500://Set home position and home flag
	IF Position <> DEFAULT_HOME_POSITION
	THEN
		MC_Home.Position									:= Position + (ABS(MemBlockPos - Axis.NcToPlc.ActPos) * SEL(MC_Velocity.Direction = MC_Negative_Direction, -1.0 , 1.0));
	ELSE
		MC_Home.Position									:= Param_CalibrationValue + (ABS(MemBlockPos - Axis.NcToPlc.ActPos) * SEL(MC_Velocity.Direction = MC_Negative_Direction, -1.0 , 1.0)); 
	END_IF
	MC_Home(
		Axis 		:= Axis,
		Execute		:= TRUE,
		Position	:= , //see above 
		HomingMode	:= MC_Direct
	);
	IF NOT MC_Home.Busy 
	THEN
		IF NOT MC_Home.Error
		THEN
			MemError										:= TRUE;
			LastErrorState									:= state;
			LastErrorId										:= MC_Absolute.ErrorID;	
			state											:= 600; //Try to restore old parameter first			
		ELSE
			state											:= 600;
		END_IF
		MC_Home(Execute := FALSE, Axis := Axis);
	END_IF

(* Return parameters for NC and drive to prior value ************************************************)
600:
	uiValue													:= TO_UINT(Param_MotionMonitoring.1);
	Write_ADS(NetId:= '' , Port:=500, IdxGrp:=16#4000+Axis.NcToPlc.AxisId, IDxOffs:=16#11,
				LEN:=SIZEOF(uiValue), SrcAddr:=ADR(uiValue), Write := Param_MotionMonitoring.0 );
	IF NOT Write_ADS.BUSY 
	THEN
		IF Write_ADS.ERR AND NOT MemError
		THEN
			MemError										:= TRUE;
			LastErrorState									:= state;
			LastErrorId										:= Write_ADS.ERRID;	
		END_IF
		Write_ADS(Write := FALSE);
		State												:= state + 1;									
	END_IF
		
601:
	uiValue													:= TO_UINT(Param_LagMonitoring.1);	
	Write_ADS(NetId:= '' , Port:=500, IdxGrp:=16#6000+Axis.NcToPlc.AxisId, IDxOffs:=16#10,
				LEN:=SIZEOF(uiValue), SrcAddr:=ADR(uiValue), Write := Param_LagMonitoring.0 );
	IF NOT Write_ADS.BUSY 
	THEN
		IF Write_ADS.ERR AND NOT MemError
		THEN
			MemError										:= TRUE;
			LastErrorState									:= state;
			LastErrorId										:= Write_ADS.ERRID;	
		END_IF
		Write_ADS(Write := FALSE);
		State												:= state + 1;									
	END_IF
	
602:
	uiValue													:= TO_UINT(Param_SoftMaxMonitoring.1);
	Write_ADS(NetId:= '' , Port:=500, IdxGrp:=16#5000+Axis.NcToPlc.AxisId, IDxOffs:=16#C,
				LEN:=SIZEOF(uiValue), SrcAddr:=ADR(uiValue), Write := Param_SoftMaxMonitoring.0 );
	IF NOT Write_ADS.BUSY 
	THEN
		IF Write_ADS.ERR AND NOT MemError
		THEN
			MemError										:= TRUE;
			LastErrorState									:= state;
			LastErrorId										:= Write_ADS.ERRID;	
		END_IF
		Write_ADS(Write := FALSE);
		State												:= state + 1;									
	END_IF
	
603:
	uiValue													:= TO_UINT(Param_SoftMinMonitoring.1);
	Write_ADS(NetId:= '' , Port:=500, IdxGrp:=16#5000+Axis.NcToPlc.AxisId, IDxOffs:=16#B,
				LEN:=SIZEOF(uiValue), SrcAddr:=ADR(uiValue), Write := Param_SoftMinMonitoring.0 );
	IF NOT Write_ADS.BUSY 
	THEN
		IF Write_ADS.ERR AND NOT MemError
		THEN
			MemError										:= TRUE;
			LastErrorState									:= state;
			LastErrorId										:= Write_ADS.ERRID;	
		END_IF
		Write_ADS(Write := FALSE);
		State												:= 604;									
	END_IF

604:
	IF DrvChannel = 1
	THEN
		CoERead.Index										:= SEL(DriveProfileIsDS402, 16#7110 , 	16#6872); 
		CoERead.SubIndex									:= SEL(DriveProfileIsDS402, 16#B  , 	16#0);
	ELSE //Channel 0
		CoERead.Index										:= SEL(DriveProfileIsDS402, 16#7010 , 	16#6072);
		CoERead.SubIndex									:= SEL(DriveProfileIsDS402, 16#B  , 	16#0);
 	END_IF 

	uiValue													:= Param_MaxTorque;
	CoEWrite(
		NetId			:= '', 
		Index			:= ,//See above
		SubIndex		:= , //See above 
		pSrcBuf			:= ADR(uiValue), 
		BufLen			:= SIZEOF(uiValue),//2,
		Execute			:= Param_MaxTorqueRead, 
		Axis			:= Axis
	);
	IF NOT CoEWrite.BUSY 
	THEN
		IF CoEWrite.Error
		THEN
			MemError										:= TRUE;
			LastErrorState									:= state;
			LastErrorId										:= CoEWrite.AdsErrId;//or CANopenErrId;				
		END_IF
		CoEWrite(Execute := FALSE, Axis := Axis);
		state												:= 900;			
	END_IF
	
(* Done *****************************************************************************)
900://Wait for execute signal to change to false
	Done 													:= NOT MemError; //Set the done flag to true if not error occur
	BUSY 													:= FALSE;
	Error													:= MemError;
	ErrorId													:= SEL(Error, 0 , LastErrorId);
	
	//Make sure all components stop operating
	Read_ADS(Read := FALSE);	Write_Ads(Write := FALSE);
	CoEWrite(Execute := FALSE,axis  := axis); CoERead(Execute := FALSE,axis  := axis);	
	MC_Home(Execute := FALSE,Axis := Axis);
	MC_Halt(Execute := FALSE,Axis := Axis);
	MC_Velocity(Execute := FALSE,Axis := Axis);
	MC_Absolute(Execute := FALSE,Axis := Axis);	
	
	State													:= 0;
END_CASE

END_FUNCTION_BLOCK

// POUs/Motion/TF50xx-NC/02_Options/Motion/AxMoveSinus
{attribute 'pack_mode' := '4'}
FUNCTION_BLOCK AxMoveSinus EXTENDS FbBase
VAR_INPUT
	Frequence												: LREAL := 0.0; //Hz
	SinusVeloAmplitude										: LREAL := 0.0; //mm/s
	DrivingTime												: TIME := T#0MS; //s
END_VAR
VAR_IN_OUT
	Axis													: AXIS_REF;
END_VAR
VAR_OUTPUT
	Active													: booL := FALSE;
	CommandAborted											: BOOL := FALSE;
END_VAR
VAR //Sinus Oscillation Sequence
(* 
- used as single sinus oscillation (sinus generator)
- used as sinus oscillation sequence (e.g. for bode plot) NEW 
UINT32 ENUM 1 				start type (fixed to start type 1 yet) 
UINT32 Reserved			
REAL64 e.g. mm/s > 0.0 		base amplitude (e.g. 2.5 mm/s) 
REAL64 Hz [0.0 .... 10.0] 	base frequency (e.g. 1.953125 Hz) 
REAL64 e.g. mm/s ≥ 0.0 		start amplitude at begin (e.g. 0.0 mm/s) 
REAL64 e.g. mm/REV > 0.0 	feed constant motor (per motor turn) (e.g. 10.0 mm/REV) 
REAL64 Hz ≥ 1.0 			frequency range: start frequency (e.g. 20.0 Hz) 
REAL64 Hz ≤ 1/(2*dT) 		frequency range: stop frequency (e.g. 500.0 Hz) 
REAL64 s > 0.0 				step duration (e.g. 2.048s) 
UINT32 1 [1 ... 200] 		number of measurements (step cycles) (e.g. 20) 
UINT32 1   					number of parallel measurements (e.g. 1)   not used yet! 
=72
*)   
	StartType												:	UDINT := TO_UDINT(Tc2_MC2._E_TCNC_StartPosType.TCNC_START_ABSOLUTE);
	Reserved												:	UDINT := 0;	
	BaseAmplitude											:	LREAL := 2.5;
	BaseFrequency											:	LREAL := 1.953125;
	StartAmplitude											:	LREAL := 0.0;
	FeedConstantMotor										:	LREAL := 10.0;
	FreqRangeStartFreq										:	LREAL := 0.0;
	FreqRangeStopFreq										:	LREAL := 500.0;								
	StepDuration											:	LREAL := 0.0;
	NumOfMeasurements										:	UDINT  := 0; //StepCount
	NumOfParallelMeasurements								:	UDINT  := 1;	
END_VAR
VAR
(* Internal memory **********************************************************************)
	LastErrorID												:	UDINT;
	StartCmdNo												: WORD;
	
(* Timer ********************************************************************************)                 	
	tonTimeout												:	TON;

(* Trigger ******************************************************************************)

(* FB instances *************************************************************************)
	Write_ADS												: ADSWRITE  := (NetId := '', Port := AMSPORT_R0_NCSAF, IdxGrp := 16#4200 + 0, IdxOffs := 16#33, LEN := 72, TmOut := DEFAULT_ADS_TIMEOUT);

(* Dummys *******************************************************************************)

END_VAR


(* Sinus Oscillation Sequence *************************************************************************************)
rtExecute(CLK := Execute);
CASE State OF
0://Wait for execute signal to change state to true
	IF NOT Execute OR rtExecute.Q	
	THEN
		Write_Ads(WRITE := FALSE);
		tonTimeout(IN := FALSE);
		FreqRangeStartFreq									:= Frequence;
		StartAmplitude										:= SinusVeloAmplitude;
		StepDuration										:= TO_LREAL(DrivingTime) * 0.001; //time ms to lreal s
		Busy												:= rtExecute.Q;
		CommandAborted										:= FALSE;
		Active												:= FALSE;
		Done 												:= FALSE;
		Error												:= FALSE;
		ErrorID												:= 0;
		StartCmdNo											:= Axis.NcToPlc.CmdNo;

		Write_ADS( //See also declaration
			IdxGrp	:=	16#4200+Axis.NcToPlc.AxisId,
			SrcAddr	:=ADR(StartType), 
			Write 	:= rtExecute.Q);
		
		state												:= SEL(Write_ADS.Write, 0, state + 1);
	
	END_IF

1://Read original parameters for position lag monitoring
	Write_ADS(SrcAddr	:=ADR(StartType)); 
	IF NOT Write_ADS.BUSY 
	THEN
		IF Write_ADS.ERR 
		THEN
			LastErrorId										:= Write_ADS.ERRID;	
			BUSY 											:= FALSE;
			Error											:= TRUE;
			ErrorId											:= LastErrorId;
			State											:= 0;
		ELSE				
			Active 											:= F_AxisHasJob(Axis.NcToPlc.StateDWord) AND StartCmdNo <> Axis.NcToPlc.CmdNo;	
			state											:= state + 1;
		END_IF
		Write_ADS(Write := FALSE);
	END_IF

2: //Wait for command done
	IF F_AxisHasJob(Axis.NcToPlc.StateDWord) AND StartCmdNo <> Axis.NcToPlc.CmdNo
	THEN
		Active												:= TRUE;
	ELSIF F_AxisInErrorState(Axis.NcToPlc.StateDWord) 
	THEN
		Active												:= FALSE;
		Busy												:= FALSE;
		(* axis error came up before this command has been started *)
		Error 												:= TRUE;
		ErrorID 											:= AXIS.NcToPlc.ErrorCode;
		LastErrorId											:= ErrorId;
		state												:= 0;
		
	ELSIF F_AxisIsCoupled(Axis.NcToPlc.CoupleState) 
		OR F_AxisHasBeenStopped(Axis.NcToPlc.StateDWord) 
	THEN
		(* if axis is coupled during motion (FlyingSaw) all commands are aborted *)
		Active												:= FALSE;
		Busy												:= FALSE;
		CommandAborted 										:= TRUE;
		state												:= 0;																																     	

	ELSIF Active
	THEN //No longer active
		Active												:= FALSE;
		Busy												:= FALSE;
		Done												:= TRUE;
		state												:= 0;		
	ELSE 	
		tonTimeOut(In := TRUE, PT := T#100MS);
		IF tonTimeOut.Q
		THEN //Command not responded
			Busy											:= FALSE;
			Error 											:= TRUE;
			ErrorID 										:= MC_ERROR_STATE_FEEDBACK_TIMEOUT;
			state											:= 0;				
		END_IF			
	END_IF
END_CASE
(********************************************************************************************)

END_FUNCTION_BLOCK

// POUs/Motion/TF50xx-NC/02_Options/Motion/AxSuperposition
FUNCTION_BLOCK AxSuperposition EXTENDS AxFbBase
VAR_OUTPUT CONSTANT 
	FNC_MOVEIMPOSED											:	INT := 0;
	FNC_MOVEABORT											:	INT := 1;
END_VAR                     								
VAR_INPUT                   								
	Fnc														:	INT := FNC_MOVEIMPOSED;
	Mode    												:	E_SuperpositionMode;
	Distance      											:	LREAL;
	VelocityDiff 											:	LREAL;
	Acc			 											:	LREAL;
	Dec			 											:	LREAL;
	Jerk    												:	LREAL;
	VelocityProcess   										:	LREAL;
	Length    												:	LREAL;
	Options    												:	ST_SuperpositionOptions;
                            							
END_VAR
VAR_IN_OUT
END_VAR
VAR_OUTPUT
	Warning													:	BOOL;
	WarningId												:	UDINT;
END_VAR
VAR
(* Zwischenspeicher ****************************************)
	MemFnc													:	INT := -1;

(* Timer ***************************************************)

(* Trigger *************************************************)

(* Instanzierung der MC Bausteine **************************)
	MC_MoveImposed											:	MC_MoveSuperImposed;
	MC_MoveAbort											:	MC_AbortSuperposition;

(* Dummy Speicher ******************************************)

END_VAR

	(************************************************************************************)
	(*																					*)
	(*		B E C K H O F F   N E W   A U T O M A T I O N   T E C H N O L O G Y    		*)
	(*																					*)
	(*		Eiserstr.5	D-33415 Verl	Germany	phone:	+49-5246-0	www.Beckhoff.com	*)
  	(*																					*)
  	(*		Bausteinbeschreibung	:	Move Imposed Achs Baustein						*)
	(*		TwinCAT-Version			:	3.1		 										*)
	(*		Version					:	V1.0 / 04/16									*)
 	(*																					*)
	(*																					*)
	(************************************************************************************)

(* Execute ******************************************************************************)
	rtExecute(CLK := Execute);
	IF rtExecute.Q
		AND MemFnc < 0
	THEN
		MemFnc 												:= Fnc ;
		Busy												:= TRUE;
		Done												:= FALSE;
		Active												:= FALSE;
		Error												:= FALSE;
		ErrorID												:= 0;
		Warning												:= FALSE;
		WarningId											:= 0;
		CmdAborted											:= FALSE;
		ErrorText											:= '';
	END_IF

(* Call Method ***********************************************************************************)
	CASE MemFnc OF
	FNC_MOVEIMPOSED:
		MoveImposed(Execute);

	FNC_MOVEABORT:
		MoveAbort(Execute);

	-1:
		IF NOT Execute
		THEN
			Busy											:= FALSE;
			Done											:= FALSE;
			Active											:= FALSE;
			Error											:= FALSE;
			ErrorID											:= 0;
			Warning											:= FALSE;
			WarningId										:= 0;
			CmdAborted										:= FALSE;
			ErrorText										:= '';
		END_IF
	ELSE
		Busy												:= FALSE;
		Done												:= FALSE;
		Active												:= FALSE;
		Error												:= Execute;
		ErrorID												:= E_AdsErr.DEVICE_INVALIDPARM;
		Warning												:= Execute;
		WarningId											:= 0;
		CmdAborted											:= FALSE;
		ErrorText											:= CONCAT('invalid parameter value(s) Fnc no: ' , INT_TO_STRING(MemFnc));
	END_CASE

(*************************************************************************************************)

METHOD PUBLIC moveAbort : BOOL //Return value = TRUE if busy
VAR_INPUT
	Execute													:	BOOL;
END_VAR
	MemFnc 													:= FNC_MOVEABORT;

IF NOT __ISVALIDREF(rAxis) 
THEN
	Busy													:= NOT Error;
	Error													:= TRUE;
	ErrorId													:= E_AdsErr.DEVICE_INVALIDPARM;
	CmdAborted												:= FALSE;
	Done													:= FALSE;
	Active													:= FALSE;
	ErrorText												:= 'Reference rAxis invalid (0)';
	MemFnc													:= SEL(Execute , -1 ,MemFnc); 
	RETURN;
END_IF


MC_MoveAbort(
	Execute													:= Execute,
	Axis													:= rAxis,
	Done													=> Done,
	Busy													=> Busy,
	Error													=> Error,
	ErrorID													=> ErrorID);

	IF Error THEN
		LastErrorId											:= ErrorID;
		ErrorText 											:= CONCAT('Error MC_MoveAbort ID:' , UDINT_TO_STRING(ErrorId));
	ELSE
		ErrorText 											:= '';
	END_IF

	IF NOT Execute AND NOT Busy
	THEN
		MemFnc												:=  -1;
	END_IF

	MoveAbort												:= Busy;
END_METHOD

METHOD PUBLIC moveImposed : BOOL //Return value = TRUE if busy
VAR_INPUT
	Execute													:	BOOL;
END_VAR
	MemFnc 													:= FNC_MOVEIMPOSED;
	
IF NOT __ISVALIDREF(rAxis) 
THEN
	Busy													:= NOT Error;
	Error													:= TRUE;
	ErrorId													:= E_AdsErr.DEVICE_INVALIDPARM;
	CmdAborted												:= FALSE;
	Done													:= FALSE;
	Active													:= FALSE;
	ErrorText												:= 'Reference rAxis invalid (0)';
	MemFnc													:= SEL(Execute , -1 ,MemFnc); 
	RETURN;
END_IF

	MC_MoveImposed(
		Execute												:= Execute,
		Mode												:= Mode,
		Distance											:= Distance,
		VelocityDiff										:= VelocityDiff,
		Acceleration										:= Acc,
		Deceleration										:= Dec,
		Jerk												:= Jerk,
		VelocityProcess										:= VelocityProcess,
		Length												:= Length,
		Options												:= Options,
		Axis												:= rAxis,
		Done												=> Done,
		Busy												=> Busy,
		Active												=> Active,
		CommandAborted										=> CmdAborted,
		Error												=> Error,
		ErrorID												=> ErrorID,
		Warning												=> Warning,
		WarningId											=> WarningID,
		ActualVelocityDiff									=> ,
		ActualDistance										=> ,
		ActualLength										=> ,
		ActualAcceleration									=> ,
		ActualDeceleration									=> );


	IF Error THEN
		LastErrorId											:= ErrorID;
		ErrorText 											:= CONCAT('Error MC_MoveSuperImposed ID:' , UDINT_TO_STRING(ErrorId));
	ELSE                            					
		ErrorText 											:= '';
	END_IF

	IF NOT Execute AND NOT Busy
	THEN
		MemFnc												:=  -1;
	END_IF

	MoveImposed												:= Busy;
END_METHOD

END_FUNCTION_BLOCK

// POUs/Motion/TF50xx-NC/02_Options/Parameter/AxParaCtrl
{attribute 'no_check'}
//FB to read and write NC axis controller parameter in particular  
//The FB can be enherided and derivatived methods of SeqRead/SeqWrite used for application specific parameter.
//The extended methods need to call the super class at the beginning and return true if execution will be finished. The allowed states for new parameter are 1..99
FUNCTION_BLOCK AxParaCtrl EXTENDS AxRWParaBase
VAR_OUTPUT CONSTANT
END_VAR                                 					
VAR_INPUT                               					                                   	                                        	
	AxisID													: 	UDINT;				(* ID der Achse *)

	(* Write *)
	SetPosLoopDeadBandPosDeviation							: 	LREAL;//Positon ctrl loop: 'dead band' in mm for position error (position deviation)(for P/PID-controller with velocity or torque interface)
	SetPosLoop_Kv											: 	LREAL;//Positon ctrl loop: Proportional amplification factor kp resp. kv (Standstill for two P-Const)
	SetPosLoop_Kv2Moving									: 	LREAL;//Positon ctrl loop: With two P-Const: Add proportional amplification factor kp resp. kv that applies above a limit velocity in percent 
	SetPosLoop_Tn											: 	LREAL;//Positon ctrl loop: Integral action time Tn in sec
	SetPosLoop_Tv											: 	LREAL;//Positon ctrl loop: Derivative action time Tv sec																			
	SetPosLoop_Td											: 	LREAL;//Positon ctrl loop: Damping time Td in sec																		
	
	SetPosLoopVeloThreshold									: 	LREAL;//Positon ctrl loop: Threshold level velocity in percent, above which the additional proportional amplification factor kp resp. kv applies.

	SetPosLoopMinMaxLimit_I_Part							: 	LREAL;//Positon ctrl loop: Min/Maximum output limitation ( ) for I- part in percent (default setting: 0.1 == 10 %)																	
	SetPosLoopMinMaxLimit_D_Part							: 	LREAL;//Positon ctrl loop: Min/Maximum output limitation ( ) for D- part in percent (default setting: 0.1 == 10 %)																
	SetPosLoopDisable_I_Part								: 	BOOL;//Positon ctrl loop: Switch off the I-part during an active positioning process (as far as I-part active)? (default setting: 0 = FALSE)										
 
	SetPosLoopFeedFwdAcc_Ka 								: 	LREAL;//Positon ctrl loop: Feed forward acceleration, proportional amplification factor Kv (Acceleration pre control)							
	SetPosLoopFeedFwdVeloPreCntrlWeight						: 	LREAL;//Positon ctrl loop: Weight of the velocity pre control (standard value: 1.0 = 100 %)
	
//Velocity control loop CtrlType 5,6)
	SetVeloLoopDeadBandVeloDeviation						: 	LREAL;//Velocity ctrl loop: 'dead band' for velocity error (velocity deviation)(for P/PID-controller with velocity or torque interface)
	SetVeloLoopFilterTimeVeloDeviation						: 	LREAL;//Velocity ctrl loop: PT-2 filter time for velocity error (velocity-difference)
                                                                         
	SetVeloLoop_Kv											: 	LREAL;//Velocity ctrl loop: The Proportional Factor Kv is the gain factor of the P-controller.
	SetVeloLoop_Tn											: 	LREAL;//Velocity ctrl loop: Integral Action Time Tn of the I component of the PID-controller in sec
	SetVeloLoop_Tv											: 	LREAL;//Velocity ctrl loop: Rate time Tv of the real D component (D-T1 component) of the PID-controller in sec																			
	SetVeloLoop_Td											: 	LREAL;//Velocity ctrl loop: Damping time Td of the real D component (D-T1 component) of the PID-controller in sec																		
                                                                         
	SetVeloLoopMinMaxLimit_D_Part							: 	LREAL;//Velocity ctrl loop: Min/Maximum output limitation ( ) for D- part in percent (default setting: 0.1 == 10 %)	
	SetVeloLoopMinMaxLimit_I_Part							: 	LREAL;//Velocity ctrl loop: Min/Maximum output limitation ( ) for I- part in percent (default setting: 0.1 == 10 %)																	

END_VAR
VAR_OUTPUT    
	CtrlType												: 	UDINT;(* Controller Type:
																			0 NOT DEFINED
																			1 Position-controller (standard) (Position)
																			2 Position-controller with two P-constants (with ka) (Position)
																			3 Position-controller PID (with ka)(Position)
																			5 Position and velocity P-controller(with ka) (Velocity)
																			6 PI controller (Velocity)
																			7 High/low speed controller (Position)
																			8 Stepper motor controller(Position)
																			9 SERCOS controller(Position in the drive)
																			10 RESERVED
																			11 RESERVED
																			12 RESERVED
																			13 RESERVED
																			14 TCom Controller (Soft Drive)(Position in the drive)*)

																		
//Position control loop
	PosLoopDeadBandPosDeviation								: 	LREAL;//Positon ctrl loop: 'dead band' in mm for position error (position deviation)(for P/PID-controller with velocity or torque interface)
	PosLoop_Kv												: 	LREAL;//Positon ctrl loop: Proportional amplification factor kp resp. kv (Standstill for two P-Const)
	PosLoop_Kv2Moving										: 	LREAL;//Positon ctrl loop: With two P-Const: Add proportional amplification factor kp resp. kv that applies above a limit velocity in percent 
	PosLoop_Tn												: 	LREAL;//Positon ctrl loop: Integral action time Tn in sec
	PosLoop_Tv												: 	LREAL;//Positon ctrl loop: Derivative action time Tv sec																			
	PosLoop_Td												: 	LREAL;//Positon ctrl loop: Damping time Td in sec																		
	
	PosLoopVeloThreshold									: 	LREAL;//Positon ctrl loop: Threshold level velocity in percent, above which the additional proportional amplification factor kp resp. kv applies.

	PosLoopMinMaxLimit_I_Part								: 	LREAL;//Positon ctrl loop: Maximum output limitation ( ) for I- part in percent (default setting: 0.1 == 10 %)																	
	PosLoopMinMaxLimit_D_Part								: 	LREAL;//Positon ctrl loop: Maximum output limitation ( ) for D- part in percent (default setting: 0.1 == 10 %)																
	PosLoopDisable_I_Part									: 	BOOL; //Positon ctrl loop: Switch off the I-part during an active positioning process (as far as I-part active)? (default setting: 0 = FALSE)										
 
	PosLoopFeedFwdAcc_Ka 									: 	LREAL;//Positon ctrl loop: Feed forward acceleration, proportional amplification factor Kv (Acceleration pre control)							
	PosLoopFeedFwdVeloPreCntrlWeight						: 	LREAL;//Positon ctrl loop: Weight of the velocity pre control (standard value: 1.0 = 100 %)

//Velocity control loop	(CtrlType 5,6)
	VeloLoopDeadBandVeloDeviation							: 	LREAL;//Velocity ctrl loop: 'dead band' for velocity error (velocity deviation)(for P/PID-controller with velocity or torque interface)
	VeloLoopFilterTimeVeloDeviation							: 	LREAL;//Velocity ctrl loop: PT-2 filter time for velocity error (velocity-difference)
                                                                          
	VeloLoop_Kv												: 	LREAL;//Velocity ctrl loop: The Proportional Factor Kv is the gain factor of the P-controller.
	VeloLoop_Tn												: 	LREAL;//Velocity ctrl loop: Integral Action Time Tn of the I component of the PID-controller in sec
	VeloLoop_Tv												: 	LREAL;//Velocity ctrl loop: Rate time Tv of the real D component (D-T1 component) of the PID-controller in sec																			
	VeloLoop_Td												: 	LREAL;//Velocity ctrl loop: Damping time Td of the real D component (D-T1 component) of the PID-controller in sec																		
                                                                         
	VeloLoopMinMaxLimit_D_Part								: 	LREAL;//Velocity ctrl loop: Min/Maximum output limitation ( ) for D- part in percent (default setting: 0.1 == 10 %)																
	VeloLoopMinMaxLimit_I_Part								: 	LREAL;//Velocity ctrl loop: Min/Maximum output limitation ( ) for I- part in percent (default setting: 0.1 == 10 %)																	
		
END_VAR                         	
VAR
(* Zwischenspeicher ************************************************************)
	
(* Deklaration Trigger **********************************************************)

(* Zeiten ******************************************************************)

(* Bausteine ***************************************************************)
	ReadAdsPara												: ADSREAD := (NetId	:= '' , Port := AMSPORT_R0_NC, TmOut	:= DEFAULT_ADS_TIMEOUT);
	WriteAdsPara											: ADSWRITE := (NetId:= '' , Port := AMSPORT_R0_NC, TmOut	:= DEFAULT_ADS_TIMEOUT);

(* Dummy Speicher **********************************************************)

END_VAR

	(************************************************************************************)
	(*																					*)
	(*		B E C K H O F F   N E W   A U T O M A T I O N   T E C H N O L O G Y    		*)
	(*																					*)
	(*		Eiserstr.5	D-33415 Verl	Germany	phone:	+49-5246-0	www.Beckhoff.Com	*)
    (*																					*)
    (*		Bausteinbeschreibung	:	Read/Write axis NC controller parameter			*)
	(*		TwinCAT-Version			:	3.x or higher									*)
	(*																					*)
	(************************************************************************************)

(* Execute ***************************************************************************************)
	Super^();			
	
(*************************************************************************************************)

PROPERTY PROTECTED deviceAddrIsValid : BOOL
GET
deviceAddrIsValid := AxisId > 0;
END_GET
END_PROPERTY

METHOD PROTECTED getValue : BOOL //Return value = TRUE if execution finished and state incremented 
VAR_INPUT
	IDxGrp						:	UDINT;
	IDxOffs						:	UDINT;
	Len							:	UDINT;
	pActValue					:	PVOID; //Address of variable for actual value
	pSetValue					:	PVOID; //Address of variable for ser value variable, can be zero if no corresponding SetVariable exists
END_VAR

ReadAdsPara	(Read := TRUE, IDxGrp:=IDxGrp+AxisId, IDxOffs:=IDxOffs,LEN:=Len,DestAddr:=pActValue );
IF NOT ReadAdsPara.BUSY
THEN
	IF NOT ReadAdsPara.ERR 
	THEN 
		IF pSetValue <> 0 THEN MEMCPY(pSetValue, pActValue, Len); END_IF			
		state 												:= state + 1; 
	ELSE 		
		Busy												:= FALSE;
		Error												:= TRUE;
		ErrorId												:= ReadAdsPara.ERRID;
		ErrorText											:= CONCAT('Error read parameter in state:' , TO_STRING(state * -1));
		ErrorText											:= CONCAT(ErrorText , ' Id:');
		ErrorText											:= CONCAT(ErrorText , TO_STRING(ErrorId));
		State												:= 9999;
	END_IF	
	ReadAdsPara(Read := FALSE); 
	getValue												:= TRUE;									
END_IF
END_METHOD

METHOD PROTECTED seqRead : BOOL //Return value = TRUE if execution finished 
VAR_IN_OUT
	State							:	INT;
END_VAR
(* Execute read axis parameter ************************************)
	CASE state OF
	1..99: //read application spec parameter 
		seqRead												:= TRUE;
		
	1001: (* Type **********************************************************************************)
		IF CtrlType <> 0 AND NOT ReadAdsPara.BUSY
		THEN
			state											:= state + 1;
		ELSE
			getValue(IDxGrp:= 16#6000,	IDxOffs := 16#3,	LEN := SIZEOF(CtrlType),	pActValue := ADR(CtrlType), 	pSetValue := 0);
		END_IF

	1002: (* Pos Ctrl loop. dead band (2,3,12,13 ****************************************************************************************)
		IF CtrlType <> 2 AND CtrlType <> 3 AND CtrlType <> 12 AND CtrlType <> 13 
		THEN
			state											:= state + 1;
		ELSE
			getValue(IDxGrp:= 16#6000,	IDxOffs := 16#10D,	LEN := SIZEOF(PosLoopDeadBandPosDeviation),	pActValue := ADR(PosLoopDeadBandPosDeviation), 	pSetValue := ADR(SetPosLoopDeadBandPosDeviation));
		END_IF

	1003: (* Pos control Kv (Standstill) (1,2,3,5,6,10,11,12,13 ****************************************************************************************)
		IF CtrlType > 6 AND CtrlType < 10 OR CtrlType > 13 
		THEN
			state											:= state + 1;
		ELSE
			getValue(IDxGrp:= 16#6000,	IDxOffs := 16#102,	LEN := SIZEOF(PosLoop_Kv),	pActValue := ADR(PosLoop_Kv), pSetValue := ADR(SetPosLoop_Kv));
		END_IF
		
	1004: (* Pos control Kv (Moving) (2, ****************************************************************************************)
		IF CtrlType <> 2 
		THEN
			state											:= state + 1;
		ELSE
			getValue(IDxGrp:= 16#6000,	IDxOffs := 16#106,	LEN := SIZEOF(PosLoop_Kv2Moving),	pActValue := ADR(PosLoop_Kv2Moving), pSetValue := ADR(SetPosLoop_Kv2Moving));
		END_IF
	
	1005: (* Pos control Integral action time Tn (3,10,11 ***********************************************************************)
		IF CtrlType <> 3 AND CtrlType <> 10 AND CtrlType <> 11
		THEN
			state											:= state + 1;
		ELSE
			getValue(IDxGrp:= 16#6000,	IDxOffs := 16#103,	LEN := SIZEOF(PosLoop_Tn),	pActValue := ADR(PosLoop_Tn),  pSetValue := ADR(SetPosLoop_Tn) );	
		END_IF
		
	1006: (* Pos control Derivative action time Tv (3,10,11 ***********************************************************************)
		IF CtrlType <> 3 AND CtrlType <> 10 AND CtrlType <> 11
		THEN
			state											:= state + 1;
		ELSE
			getValue(IDxGrp:= 16#6000,	IDxOffs := 16#104,	LEN := SIZEOF(PosLoop_Tv),	pActValue := ADR(PosLoop_Tv),  pSetValue := ADR(SetPosLoop_Tv) );
		END_IF
		
	1007: (* Pos control Damping time Td (3,10,11 ***************************************************************)
		IF CtrlType <> 3 AND CtrlType <> 10 AND CtrlType <> 11 
		THEN
			state											:= state + 1;
		ELSE
			getValue(IDxGrp:= 16#6000,	IDxOffs := 16#105,	LEN := SIZEOF(PosLoop_Td),	pActValue := ADR(PosLoop_Td), pSetValue := ADR(PosLoop_Td));
		END_IF

	1008: (* Pos control with 2 P-Const, Threshold level velocity in percent (2,) ***************************************************************)
		IF CtrlType <> 2 
		THEN
			state											:= state + 1;
		ELSE
			getValue(IDxGrp:= 16#6000,	IDxOffs := 16#107,	LEN := SIZEOF(PosLoopVeloThreshold),	pActValue := ADR(PosLoopVeloThreshold), pSetValue := ADR(SetPosLoopVeloThreshold));
		END_IF
		
	1009: (* Pos control Maximum output limitation ( ) for I- part in percent (3,10,11 ***************************************************************)
		IF CtrlType <> 3 AND CtrlType <> 10 AND CtrlType <> 11
		THEN
			state											:= state + 1;
		ELSE
			getValue(IDxGrp:= 16#6000,	IDxOffs := 16#116,	LEN := SIZEOF(PosLoopMinMaxLimit_I_Part),	pActValue := ADR(PosLoopMinMaxLimit_I_Part), pSetValue := ADR(SetPosLoopMinMaxLimit_I_Part));
		END_IF
		
	1010: (* Pos control Maximum output limitation ( ) for D- part in percent (3,10,11 ***************************************************************)
		IF CtrlType <> 3 AND CtrlType <> 10 AND CtrlType <> 11
		THEN
			state											:= state + 1;
		ELSE
			getValue(IDxGrp:= 16#6000,	IDxOffs := 16#117,	LEN := SIZEOF(PosLoopMinMaxLimit_D_Part),	pActValue := ADR(PosLoopMinMaxLimit_D_Part), pSetValue := ADR(SetPosLoopMinMaxLimit_D_Part));
		END_IF		

	1011: (* Pos control Switch off the I-part during an active positioning process (3,)***************************************************************)
		IF CtrlType <> 3 
		THEN
			state											:= state + 1;
		ELSIF getValue(IDxGrp:= 16#6000,	IDxOffs := 16#118,	LEN := SIZEOF(_UINT),	pActValue := ADR(_UINT),  pSetValue := 0)
		THEN
			SetPosLoopDisable_I_Part :=PosLoopDisable_I_Part := TO_BOOL(_UINT);
		END_IF
	
	1012:(* Pos control Feed forward acceleration (1,2,3,5,6,10,11,12,13 ***************************************************************)
		IF CtrlType > 6 AND CtrlType < 10 OR CtrlType > 13 
		THEN
			state											:= state + 1;
		ELSE
			getValue(IDxGrp:= 16#6000,	IDxOffs := 16#108,	LEN := SIZEOF(PosLoopFeedFwdAcc_Ka),	pActValue := ADR(PosLoopFeedFwdAcc_Ka), pSetValue := ADR(SetPosLoopFeedFwdAcc_Ka));
		END_IF	

	1013:(* Pos control Weight of the velocity pre contr *(1,2,3,5,6,10,11,12,13,14,..)  **************************************************************)
		getValue(IDxGrp:= 16#6000,	IDxOffs := 16#B,	LEN := SIZEOF(PosLoopFeedFwdVeloPreCntrlWeight),	pActValue := ADR(PosLoopFeedFwdVeloPreCntrlWeight), pSetValue := ADR(SetPosLoopFeedFwdVeloPreCntrlWeight));

//Velocity control 
	1014:(* Velocity control dead band velocity deviation (12, ***************************************************************)
		IF CtrlType <> 12
		THEN
			state											:= state + 1;
		ELSE
			getValue(IDxGrp:= 16#6000,	IDxOffs := 16#20D,	LEN := SIZEOF(VeloLoopDeadBandVeloDeviation),	pActValue := ADR(VeloLoopDeadBandVeloDeviation), pSetValue := ADR(SetVeloLoopDeadBandVeloDeviation));
		END_IF	
		
	1015:(* Velocity control Filter time velocity deviation (12, ***************************************************************)
		IF CtrlType <> 12
		THEN
			state											:= state + 1;
		ELSE
			getValue(IDxGrp:= 16#6000,	IDxOffs := 16#220,	LEN := SIZEOF(VeloLoopFilterTimeVeloDeviation),	pActValue := ADR(VeloLoopFilterTimeVeloDeviation), pSetValue := ADR(SetVeloLoopFilterTimeVeloDeviation));
		END_IF			
		
	1016:(* Velocity control: Proportional Factor Kv (5,6,12,13 ***************************************************************)
		IF CtrlType <> 5 AND CtrlType <> 6 AND CtrlType <> 12 AND CtrlType <> 13
		THEN
			state											:= state + 1;
		ELSE
			getValue(IDxGrp:= 16#6000,	IDxOffs := 16#202,	LEN := SIZEOF(VeloLoop_Kv),	pActValue := ADR(VeloLoop_Kv), pSetValue := ADR(SetVeloLoop_Kv));
		END_IF		
	
   	1017:(* Velocity control: Integral Action Time Tn (6,12***************************************************************)
		IF CtrlType <> 6 AND CtrlType <> 12
		THEN
			state											:= state + 1;
		ELSE
			getValue(IDxGrp:= 16#6000,	IDxOffs := 16#203,	LEN := SIZEOF(VeloLoop_Tn),	pActValue := ADR(VeloLoop_Tn), pSetValue := ADR(SetVeloLoop_Tn));
		END_IF										

   	1018:(* Velocity control: Derivative Action Time Tv (6,12 ***************************************************************)
		IF CtrlType <> 6 AND CtrlType <> 12
		THEN
			state											:= state + 1;
		ELSE
			getValue(IDxGrp:= 16#6000,	IDxOffs := 16#204,	LEN := SIZEOF(VeloLoop_Tv),	pActValue := ADR(VeloLoop_Tv), pSetValue := ADR(SetVeloLoop_Tv));
		END_IF	
		
   	1019:(* Velocity control: Damping Time Td (6,12 ***************************************************************)
		IF CtrlType <> 6 AND CtrlType <> 12
		THEN
			state											:= state + 1;
		ELSE
			getValue(IDxGrp:= 16#6000,	IDxOffs := 16#205,	LEN := SIZEOF(VeloLoop_Td),	pActValue := ADR(VeloLoop_Td), pSetValue := ADR(SetVeloLoop_Td));
		END_IF	
		
   	1020:(* Velocity control Min/Max limit I Part (6,12,13 ***************************************************************)
		IF CtrlType <> 6 AND CtrlType <> 12 AND CtrlType <> 13
		THEN
			state											:= state + 1;
		ELSE
			getValue(IDxGrp:= 16#6000,	IDxOffs := 16#206,	LEN := SIZEOF(VeloLoopMinMaxLimit_I_Part),	pActValue := ADR(VeloLoopMinMaxLimit_I_Part), pSetValue := ADR(SetVeloLoopMinMaxLimit_I_Part));
		END_IF	

   	1021:(* Velocity Min/max limit D Part (6,12 ***************************************************************)
		IF CtrlType <> 6 AND CtrlType <> 12
		THEN
			state											:= state + 1;
		ELSE
			getValue(IDxGrp:= 16#6000,	IDxOffs := 16#207,	LEN := SIZEOF(VeloLoopMinMaxLimit_D_Part),	pActValue := ADR(VeloLoopMinMaxLimit_D_Part), pSetValue := ADR(SetVeloLoopMinMaxLimit_D_Part));
		END_IF	
			
	ELSE
		state												:= 1;
	END_CASE

(*********************************************************************************************)
END_METHOD

METHOD PROTECTED seqWrite : BOOL //Return value = TRUE if execution finished 
VAR_IN_OUT
	State							:	INT;
END_VAR
(* Write axis parameter ********************************************************************)
	CASE state OF
	1..99: //Wite application spec parameter 
		seqWrite											:= TRUE;
			
	1001: (* Pos Ctrl loop. dead band  ****************************************************************************************)
		IF CtrlType <> 2 AND CtrlType <> 3 AND CtrlType <> 12 AND CtrlType <> 13 
		THEN
			state											:= state + 1;
		ELSE
			setValue(IDxGrp:= 16#6000,	IDxOffs := 16#10D,	LEN := SIZEOF(PosLoopDeadBandPosDeviation),	pActValue := ADR(PosLoopDeadBandPosDeviation), 	pSetValue := ADR(SetPosLoopDeadBandPosDeviation));
		END_IF

	1002: (* Pos control Kv (Standstill) ****************************************************************************************)
		IF CtrlType > 6 AND CtrlType < 10 OR CtrlType > 13 
		THEN
			state											:= state + 1;
		ELSE
			setValue(IDxGrp:= 16#6000,	IDxOffs := 16#102,	LEN := SIZEOF(PosLoop_Kv),	pActValue := ADR(PosLoop_Kv), pSetValue := ADR(SetPosLoop_Kv));
		END_IF
		
	1003: (* Pos control Kv (Moving) ****************************************************************************************)
		IF CtrlType <> 2 
		THEN
			state											:= state + 1;
		ELSE
			setValue(IDxGrp:= 16#6000,	IDxOffs := 16#106,	LEN := SIZEOF(PosLoop_Kv2Moving),	pActValue := ADR(PosLoop_Kv2Moving), pSetValue := ADR(SetPosLoop_Kv2Moving));
		END_IF
	
	1004: (* Pos control Integral action time Tn ***********************************************************************)
		IF CtrlType <> 3 AND CtrlType <> 10 AND CtrlType <> 11
		THEN
			state											:= state + 1;
		ELSE
			setValue(IDxGrp:= 16#6000,	IDxOffs := 16#103,	LEN := SIZEOF(PosLoop_Tn),	pActValue := ADR(PosLoop_Tn),  pSetValue := ADR(SetPosLoop_Tn) );	
		END_IF
		
	1005: (* Pos control Derivative action time Tv ***********************************************************************)
		IF CtrlType <> 3 AND CtrlType <> 10 AND CtrlType <> 11
		THEN
			state											:= state + 1;
		ELSE
			setValue(IDxGrp:= 16#6000,	IDxOffs := 16#104,	LEN := SIZEOF(PosLoop_Tv),	pActValue := ADR(PosLoop_Tv),  pSetValue := ADR(SetPosLoop_Tv) );
		END_IF
		
	1006: (* Pos control Damping time Td ***************************************************************)
		IF CtrlType <> 3 AND CtrlType <> 10 AND CtrlType <> 11
		THEN
			state											:= state + 1;
		ELSE
			setValue(IDxGrp:= 16#6000,	IDxOffs := 16#105,	LEN := SIZEOF(PosLoop_Td),	pActValue := ADR(PosLoop_Td), pSetValue := ADR(PosLoop_Td));
		END_IF

	1007: (* Pos control with 2 P-Const, Threshold level velocity in percent ***************************************************************)
		IF CtrlType <> 2 
		THEN
			state											:= state + 1;
		ELSE
			setValue(IDxGrp:= 16#6000,	IDxOffs := 16#107,	LEN := SIZEOF(PosLoopVeloThreshold),	pActValue := ADR(PosLoopVeloThreshold), pSetValue := ADR(SetPosLoopVeloThreshold));
		END_IF
		
	1008: (* Pos control Maximum output limitation ( ) for I- part in percent ***************************************************************)
		IF CtrlType <> 3 AND CtrlType <> 10 AND CtrlType <> 11
		THEN
			state											:= state + 1;
		ELSE
			setValue(IDxGrp:= 16#6000,	IDxOffs := 16#116,	LEN := SIZEOF(PosLoopMinMaxLimit_I_Part),	pActValue := ADR(PosLoopMinMaxLimit_I_Part), pSetValue := ADR(SetPosLoopMinMaxLimit_I_Part));
		END_IF
		
	1009: (* Pos control Maximum output limitation ( ) for D- part in percent ***************************************************************)
		IF CtrlType <> 3 AND CtrlType <> 10 AND CtrlType <> 11
		THEN
			state											:= state + 1;
		ELSE
			setValue(IDxGrp:= 16#6000,	IDxOffs := 16#117,	LEN := SIZEOF(PosLoopMinMaxLimit_D_Part),	pActValue := ADR(PosLoopMinMaxLimit_D_Part), pSetValue := ADR(SetPosLoopMinMaxLimit_D_Part));
		END_IF		

	1010: (* Pos control Switch off the I-part during an active positioning process ***************************************************************)
		IF NOT (SetPosLoopDisable_I_Part XOR PosLoopDisable_I_Part)
			AND NOT WriteAdsPara.BUSY
			OR CtrlType <> 3 
		THEN 
			state 											:= state + 1;
		ELSE
			_UINT											:= TO_UINT(SetPosLoopDisable_I_Part);
			PosLoopDisable_I_Part							:= SetPosLoopDisable_I_Part;
			setValue(IDxGrp:= 16#6000,	IDxOffs := 16#118,	LEN := SIZEOF(_UINT),		pActValue := 0,		pSetValue := ADR(_UINT));
		END_IF
		
	
	1011:(* Pos control Feed forward acceleration ***************************************************************)
		IF CtrlType > 6 AND CtrlType < 10 OR CtrlType > 13 
		THEN
			state											:= state + 1;
		ELSE
			setValue(IDxGrp:= 16#6000,	IDxOffs := 16#108,	LEN := SIZEOF(PosLoopFeedFwdAcc_Ka),	pActValue := ADR(PosLoopFeedFwdAcc_Ka), pSetValue := ADR(SetPosLoopFeedFwdAcc_Ka));
		END_IF	

	1012:(* Pos control Weight of the velocity pre contr ***************************************************************)
		setValue(IDxGrp:= 16#6000,	IDxOffs := 16#B,	LEN := SIZEOF(PosLoopFeedFwdVeloPreCntrlWeight),pActValue := ADR(PosLoopFeedFwdVeloPreCntrlWeight),	pSetValue := ADR(SetPosLoopFeedFwdVeloPreCntrlWeight));
		
//Velocity control 
	1013:(* Velocity control dead band velocity deviation ***************************************************************)
		IF CtrlType <> 12
		THEN
			state											:= state + 1;
		ELSE
			setValue(IDxGrp:= 16#6000,	IDxOffs := 16#20D,	LEN := SIZEOF(VeloLoopDeadBandVeloDeviation),	pActValue := ADR(VeloLoopDeadBandVeloDeviation), pSetValue := ADR(SetVeloLoopDeadBandVeloDeviation));
		END_IF	
		
	1014:(* Velocity control Filter time velocity deviation ***************************************************************)
		IF CtrlType <> 12
		THEN
			state											:= state + 1;
		ELSE
			setValue(IDxGrp:= 16#6000,	IDxOffs := 16#220,	LEN := SIZEOF(VeloLoopFilterTimeVeloDeviation),	pActValue := ADR(VeloLoopFilterTimeVeloDeviation), pSetValue := ADR(SetVeloLoopFilterTimeVeloDeviation));
		END_IF			
		
	1015:(* Velocity control: Proportional Factor Kv ***************************************************************)
		IF CtrlType <> 5 AND CtrlType <> 6 AND CtrlType <> 12 AND CtrlType <> 13
		THEN
			state											:= state + 1;
		ELSE
			setValue(IDxGrp:= 16#6000,	IDxOffs := 16#202,	LEN := SIZEOF(VeloLoop_Kv),	pActValue := ADR(VeloLoop_Kv), pSetValue := ADR(SetVeloLoop_Kv));
		END_IF		
	
   	1016:(* Velocity control: Integral Action Time Tn ***************************************************************)
		IF CtrlType <> 6 AND CtrlType <> 12
		THEN
			state											:= state + 1;
		ELSE
			setValue(IDxGrp:= 16#6000,	IDxOffs := 16#203,	LEN := SIZEOF(VeloLoop_Tn),	pActValue := ADR(VeloLoop_Tn), pSetValue := ADR(SetVeloLoop_Tn));
		END_IF										

   	1017:(* Velocity control: Derivative Action Time Tv ***************************************************************)
		IF  CtrlType <> 6 AND CtrlType <> 12
		THEN
			state											:= state + 1;
		ELSE
			setValue(IDxGrp:= 16#6000,	IDxOffs := 16#204,	LEN := SIZEOF(VeloLoop_Tv),	pActValue := ADR(VeloLoop_Tv), pSetValue := ADR(SetVeloLoop_Tv));
		END_IF	
		
   	1018:(* Velocity control: Damping Time Td ***************************************************************)
		IF CtrlType <> 6 AND CtrlType <> 12
		THEN
			state											:= state + 1;
		ELSE
			setValue(IDxGrp:= 16#6000,	IDxOffs := 16#205,	LEN := SIZEOF(VeloLoop_Td),	pActValue := ADR(VeloLoop_Td), pSetValue := ADR(SetVeloLoop_Td));
		END_IF	
		
   	1019:(* Velocity control Min/Max limit I Part ***************************************************************)
		IF CtrlType <> 6 AND CtrlType <> 12 AND CtrlType <> 13
		THEN
			state											:= state + 1;
		ELSE
			setValue(IDxGrp:= 16#6000,	IDxOffs := 16#206,	LEN := SIZEOF(VeloLoopMinMaxLimit_I_Part),	pActValue := ADR(VeloLoopMinMaxLimit_I_Part), pSetValue := ADR(SetVeloLoopMinMaxLimit_I_Part));
		END_IF	

   	1020:(* Velocity Min/max limit D Part ***************************************************************)
		IF CtrlType <> 6 AND CtrlType <> 12
		THEN
			state											:= state + 1;
		ELSE
			setValue(IDxGrp:= 16#6000,	IDxOffs := 16#207,	LEN := SIZEOF(VeloLoopMinMaxLimit_D_Part),	pActValue := ADR(VeloLoopMinMaxLimit_D_Part), pSetValue := ADR(SetVeloLoopMinMaxLimit_D_Part));
		END_IF	

	ELSE
		state 												:= 1 ;
	END_CASE
	
(***********************************************************************************************)
END_METHOD

METHOD PROTECTED setValue : BOOL //Return value = TRUE if execution finished and state incremented 
VAR_INPUT
	IDxGrp						:	UDINT;
	IDxOffs						:	UDINT;
	Len							:	UDINT;
	pActValue					:	PVOID; //Address of variable for actual value, can be zero if no corresponding acual value variable exists
	pSetValue					:	PVOID; //Address of variable for set value variable
END_VAR

IF pActValue <> 0 AND pSetValue <> 0 AND_THEN MEMCMP(pSetValue, pActValue, Len) = 0
THEN //Skip write parameter if set and actual value are equel
	state													:= state + 1;	
	setValue												:= TRUE;
ELSE
	WriteAdsPara( Write := TRUE, IdxGrp :=IDxGrp+AxisId, IdxOffs:=IDxOffs, LEN:=Len, SrcAddr:=pSetValue );
	IF NOT WriteAdsPara.BUSY
	THEN
		IF NOT WriteAdsPara.ERR
		THEN
			IF pActValue <> 0 THEN MEMCPY(pActValue, pSetValue, Len); END_IF	
			state											:= state + 1;
		ELSE
			Busy											:= FALSE;
			Error											:= TRUE;
			ErrorId											:= WriteAdsPara.ERRID;
			ErrorText										:= CONCAT('Error write parameter in state:' , TO_STRING(state * -1));
			ErrorText										:= CONCAT(ErrorText , ' Id:');
			ErrorText										:= CONCAT(ErrorText , TO_STRING(ErrorId));
			State											:= 9999;
		END_IF
		WriteAdsPara (Write := FALSE);
		setValue											:= TRUE;
	END_IF		
END_IF
END_METHOD

END_FUNCTION_BLOCK

// POUs/Motion/TF50xx-NC/02_Options/Phasing/AxPhasing
{attribute 'no_check'}
//Nc-axis phasing control 
//based on Tc2_MC2 library
FUNCTION_BLOCK AxPhasing EXTENDS AxFbBase
VAR_OUTPUT CONSTANT
	FNC_HALT_PHASING										:	INT := 0;
	FNC_PHASING_ABSOULTE									:	INT := 1;
	FNC_PHASING_RELATIVE									:	INT := 2;
END_VAR               
VAR_INPUT								
	Fnc														:	INT (FNC_HALT_PHASING..FNC_PHASING_RELATIVE) := FNC_HALT_PHASING;
	PhaseShift												:	LREAL := 0;
	Velo													:	LREAL := 0;
	Acc														:	LREAL := 0.0; // if Acc = 0, the NC-Value will be set                        								
	Dec														:	LREAL := 0.0; // if Dec = 0, the NC-Value will be set
	Jerk													:	LREAL := 0.0; // if Jerk = 0, the NC-Value will be set
	BufferMode												:	MC_BufferMode := MC_Aborting;(* 	MC_Aborting,
																									MC_Buffered,
																									MC_BlendingLow,
																									MC_BlendingPrevious,
																									MC_BlendingNext,
																									MC_BlendingHigh *)
                            								                        								
	Options 												: 	ST_PhasingOptions;
	rMasterAxis												:	REFERENCE TO AXIS_REF := 0;
END_VAR                     								
VAR_IN_OUT                  								
END_VAR                     									
VAR_OUTPUT                  	
	AbsolutePhaseShift										:	LREAL;
	CoveredPhaseShift										:	LREAL;
END_VAR
VAR
(* Zwischenspeicher **************************************************************************)
	MemFnc													:	INT := -1;

(* Trigger *)

(* Instanzierung der MC Bausteine *******************************************************)
	MC_HaltPhasing											:	MC_HaltPhasing;
	MC_PhasingAbsolute										:	MC_PhasingAbsolute;
	MC_PhasingRelative										:	MC_PhasingRelative;

(* Dummy Speicher **********************************************************)
(*	i,j		: INT := 0 ; *)
END_VAR

	(************************************************************************************)
	(*																					*)
	(*		B E C K H O F F   N E W   A U T O M A T I O N   T E C H N O L O G Y    		*)
	(*																					*)
	(*		Eiserstr.5	D-33415 Verl	Germany	phone:	+49-5246-0	www.Beckhoff.Com	*)
    (*																					*)
    (*		Bausteinbeschreibung	:	Gear axis function-block						*)
	(*		TwinCAT-Version			:	3.x or higher		 							*)
	(*		Version					:	V1.0 / 04/16									*)
 	(*		Autor					:	Thorsten Hemel									*)
	(*																					*)
	(************************************************************************************)

(* Execute ***************************************************************************************)
	rtExecute(CLK := Execute);
	IF rtExecute.Q
		AND MemFnc < 0
	THEN
		MemFnc 												:= Fnc ;
		Busy												:= TRUE;
		Done												:= FALSE;
		Active												:= FALSE;
		Error												:= FALSE;
		ErrorID												:= 0;
		CmdAborted											:= FALSE;
		ErrorText											:= '';
	END_IF

(* Call Method ***********************************************************************************)
	CASE MemFnc OF
	FNC_HALT_PHASING:
		HaltPhasing(Execute);

	FNC_PHASING_ABSOULTE:
		PhasingAbsoulte(Execute);

	FNC_PHASING_RELATIVE:
		PhasingRelative(Execute);

	-1:
		IF NOT Execute
		THEN
			Busy											:= FALSE;
			Done											:= FALSE;
			Active											:= FALSE;
			Error											:= FALSE;
			ErrorID											:= 0;
			CmdAborted										:= FALSE;
			ErrorText										:= '';
		END_IF                              				
	ELSE                                    				
		Busy												:= FALSE;
		Done												:= FALSE;
		Active												:= FALSE;
		Error												:= Execute;
		ErrorID												:= E_AdsErr.DEVICE_INVALIDPARM;
		CmdAborted											:= FALSE;
		ErrorText											:= CONCAT('invalid parameter value(s) Fnc no: ' , INT_TO_STRING(MemFnc));
	END_CASE                            		
                                            	

(*************************************************************************************************)

METHOD PUBLIC haltPhasing : BOOL //Return value = TRUE if busy
//required parameter
//rAxis
//rMasterAxis1
//RatioNumerator
//RatioDenominator
//Acc
//Dec
//Jerk
VAR_INPUT
	Execute													:	BOOL;
END_VAR
MemFnc 														:= FNC_HALT_PHASING;
THIS^.Execute												:= Execute;

IF NOT __ISVALIDREF(rAxis) 
THEN
	Busy													:= NOT Error;
	Error													:= TRUE;
	ErrorId													:= E_AdsErr.DEVICE_INVALIDPARM;
	CmdAborted												:= FALSE;
	Done													:= FALSE;
	Active													:= FALSE;
	ErrorText												:= 'Reference rAxis invalid (0)';
	MemFnc													:= SEL(Execute , -1 ,MemFnc); 
	RETURN;
ELSIF NOT __ISVALIDREF(rMasterAxis)
THEN
	Busy													:= NOT Error;
	Error													:= TRUE;
	ErrorId													:= E_AdsErr.DEVICE_INVALIDPARM;
	CmdAborted												:= FALSE;
	Done													:= FALSE;
	ErrorText												:= 'Reference rMasterAxis invalid (0)';
	MemFnc													:= SEL(Execute , -1 ,MemFnc); 
	RETURN;
END_IF

	MC_HaltPhasing(
		Execute				:= Execute, 
		Master				:= rMasterAxis, 
		Slave				:= rAxis, 
		Deceleration		:= Dec, 
		Jerk				:= Jerk, 
		BufferMode			:= BufferMode, 
		Options				:= Options, 
		Done				=> Done, 
		Busy				=> Busy, 
		Active				=> Active, 
		CommandAborted		=> CmdAborted, 
		Error				=> Error, 
		ErrorID				=> ErrorID);

	IF Error THEN
		LastErrorId											:= ErrorID;
		ErrorText 											:= CONCAT('Error MC_HaltPhasing ID:' , UDINT_TO_STRING(ErrorId));
	ELSE
		ErrorText 											:= '';
	END_IF

	IF NOT Execute AND NOT Busy
	THEN
		MemFnc												:=  -1;
	END_IF
	
	haltPhasing												:= Busy;
END_METHOD

METHOD PUBLIC phasingAbsoulte : BOOL //Return value = TRUE if busy
//required parameter
//rAxis
//rMasterAxis
//PhaseShift
//Acc
VAR_INPUT
	Execute													:	BOOL;
END_VAR
MemFnc 														:= FNC_PHASING_ABSOULTE;
THIS^.Execute												:= Execute;

IF NOT __ISVALIDREF(rAxis) 
THEN
	Busy													:= NOT Error;
	Error													:= TRUE;
	ErrorId													:= E_AdsErr.DEVICE_INVALIDPARM;
	CmdAborted												:= FALSE;
	Done													:= FALSE;
	Active													:= FALSE;
	ErrorText												:= 'Reference rAxis invalid (0)';
	MemFnc													:= SEL(Execute , -1 ,MemFnc); 
	RETURN;
ELSIF NOT __ISVALIDREF(rMasterAxis)
THEN
	Busy													:= NOT Error;
	Error													:= TRUE;
	ErrorId													:= E_AdsErr.DEVICE_INVALIDPARM;
	CmdAborted												:= FALSE;
	Done													:= FALSE;
	ErrorText												:= 'Reference rMasterAxis1 invalid (0)';
	MemFnc													:= SEL(Execute , -1 ,MemFnc); 
	RETURN;
END_IF

	MC_PhasingAbsolute(
		Execute				:= Execute, 
		Master				:= rMasterAxis, 
		Slave				:= rAxis, 
		PhaseShift			:= PhaseShift, 
		Velocity			:= Velo, 
		Acceleration		:= Acc, 
		Deceleration		:= Dec, 
		Jerk				:= Jerk, 
		BufferMode			:= BufferMode, 
		Options				:= Options, 
		Done				=> Done, 
		Busy				=> Busy, 
		Active				=> Active, 
		CommandAborted		=> CmdAborted, 
		Error				=> Error, 
		ErrorID				=> ErrorId, 
		AbsolutePhaseShift	=> AbsolutePhaseShift);
		

	IF Error THEN
		LastErrorId											:= ErrorID;
		ErrorText 											:= CONCAT('Error MC_PhasingAbsolute ID:' , UDINT_TO_STRING(ErrorId));
	ELSE
		ErrorText 											:= '';
	END_IF

	IF NOT Execute AND NOT Busy
	THEN
		MemFnc												:=  -1;
	END_IF
	
	phasingAbsoulte											:= Busy;
END_METHOD

METHOD PUBLIC phasingRelative : BOOL//Return value = TRUE if busy
//required parameter
//rAxis
//rMasterAxis
//PhaseShift
//Acc
VAR_INPUT
	Execute													:	BOOL;
END_VAR
MemFnc														:= FNC_PHASING_RELATIVE;
THIS^.Execute												:= Execute;
	                										
IF NOT __ISVALIDREF(rAxis) 
THEN
	Busy													:= NOT Error;
	Error													:= TRUE;
	ErrorId													:= E_AdsErr.DEVICE_INVALIDPARM;
	CmdAborted												:= FALSE;
	Done													:= FALSE;
	Active													:= FALSE;
	ErrorText												:= 'Reference rAxis invalid (0)';
	MemFnc													:= SEL(Execute , -1 ,MemFnc); 
	RETURN;
ELSIF NOT __ISVALIDREF(rMasterAxis)
THEN
	Busy													:= NOT Error;
	Error													:= TRUE;
	ErrorId													:= E_AdsErr.DEVICE_INVALIDPARM;
	CmdAborted												:= FALSE;
	Done													:= FALSE;
	ErrorText												:= 'Reference rMasterAxis invalid (0)';
	MemFnc													:= SEL(Execute , -1 ,MemFnc); 
	RETURN;	
END_IF
	

	MC_PhasingRelative( 
		Execute				:= Execute,
		Master				:= rMasterAxis, 
		Slave				:= rAxis, 
		PhaseShift			:= PhaseShift, 
		Velocity			:= Velo, 
		Acceleration		:= Acc, 
		Deceleration		:= Dec, 
		Jerk				:= Jerk, 
		BufferMode			:= BufferMode, 
		Options				:= Options, 
		Done				=> Done, 
		Busy				=> Busy, 
		Active				=> Active, 
		CommandAborted		=> CmdAborted, 
		Error				=> Error, 
		ErrorID				=> ErrorId, 
		CoveredPhaseShift	=> CoveredPhaseShift);					

	IF Error THEN
		LastErrorId											:= ErrorID;
		ErrorText 											:= CONCAT('Error MC_PhasingRelative ID:' , UDINT_TO_STRING(ErrorId));
	ELSE
		ErrorText 											:= '';
	END_IF

	IF NOT Execute AND NOT Busy
	THEN
		MemFnc												:=  -1;
	END_IF
	
	phasingRelative												:= Busy;
END_METHOD

END_FUNCTION_BLOCK

// POUs/Motion/TF50xx-NC/02_Options/TouchProbe/AxTouchProbe
{attribute 'no_check'}
//Nc-axis touch probe  
//based on Tc2_MC2 library
FUNCTION_BLOCK AxTouchProbe EXTENDS AxFbBase
VAR_OUTPUT CONSTANT
	FNC_RUN													:	INT := 0;
	FNC_ABORT												:	INT := 1;
END_VAR                     								
VAR_INPUT                   								
	Fnc														: 	INT (FNC_RUN..FNC_ABORT):= FNC_RUN;
	TriggerInput											: 	TRIGGER_REF;
	WindowOnly												: 	BOOL := FALSE;(* Enables the monitoring window *)
	FirstPosition											: 	LREAL;	(* Beginning of the monitoring window *)
	LastPosition 											: 	LREAL;	(* Ending of the monitoring window *)
END_VAR
VAR_IN_OUT
END_VAR
VAR_OUTPUT
	RecordedPosition										: 	LREAL;	// current axisposition on trigger-event
	RecordedData											:	MC_TouchProbeRecordedData;
END_VAR
VAR
(* cache **************************************************************************)
	MemFnc													:	INT := -1;
               								                           	
(* trigger *)               	

(* MC-function-block instances ****************************************************)
	MC_TouchProbe											: 	MC_TouchProbe;
	MC_AbortTrigger											:	MC_AbortTrigger;

END_VAR

	(************************************************************************************)
	(*																					*)
	(*		B E C K H O F F   N E W   A U T O M A T I O N   T E C H N O L O G Y    		*)
	(*																					*)
	(*		Eiserstr.5	D-33415 Verl	Germany	phone:	+49-5246-0	www.Beckhoff.Com	*)
    (*																					*)
    (*		Bausteinbeschreibung	:	TouchProbe ctrl									*)
	(*		TwinCAT-Version			:	3.x or higher 									*)
	(*		Version					:	V3.0 / 03/13									*)
	(*		Lib						:	TcMC2.lib 										*)
 	(*		Autor					:	DSC												*)
	(*																					*)
	(************************************************************************************)

(* Execute ***************************************************************************************)
	rtExecute(CLK := Execute);
	IF rtExecute.Q
		AND MemFnc < 0
	THEN
		MemFnc 												:= SEL(Fnc = FNC_RUN, FNC_ABORT , FNC_RUN) ;
		Busy												:= TRUE;
		Done												:= FALSE;
		Error												:= FALSE;
		ErrorID												:= 0;
		CmdAborted											:= FALSE;
	END_IF

(* Call Method ***********************************************************************************)
	CASE MemFnc OF
	FNC_RUN:
		Run(Execute);

	FNC_ABORT:
		Abort(Execute);

	-1:
		IF NOT Execute
		THEN
			Busy											:= FALSE;
			Done											:= FALSE;
			Error											:= FALSE;
			ErrorID											:= 0;
			CmdAborted										:= FALSE;
		END_IF                              				
	ELSE                                    				
		Busy												:= FALSE;
		Done												:= FALSE;
		Error												:= Execute;
		ErrorID												:= E_AdsErr.DEVICE_INVALIDPARM;
		CmdAborted											:= FALSE;
	END_CASE                                	

(*************************************************************************************************)

METHOD PUBLIC abort : BOOL //Return value = TRUE if busy
//required parameter
//rAxis
//TriggerInput
VAR_INPUT
	Execute													:	BOOL := FALSE;
END_VAR
	MemFnc	 												:= FNC_ABORT;
	THIS^.Execute											:= Execute;
IF NOT __ISVALIDREF(rAxis) 
THEN
	Busy													:= NOT Error;
	ErrorId													:= E_AdsErr.DEVICE_INVALIDPARM;
	Error													:= TRUE;
	Done													:= FALSE;
	CmdAborted												:= FALSE;
	MemFnc													:= SEL(Execute , -1 ,MemFnc); 
	RETURN;
END_IF

	MC_AbortTrigger(
		Execute		:= Execute,
		Axis		:= rAxis,
		TriggerInput:= TriggerInput,
		Done		=> done,
		Busy		=> Busy,
		Error		=> Error,
		ErrorID		=> ErrorID);

	CmdAborted		:= FALSE;

	IF NOT Execute AND NOT Busy
	THEN
		MemFnc												:= -1;
	END_IF                              					
	                                    	
	abort 													:= Busy;
END_METHOD

METHOD PUBLIC run : BOOL //Return value = TRUE if busy
//required parameter
//rAxis
//TriggerInput
//WindowOnly
//FirstPosition
//LastPosition
VAR_INPUT
	Execute													: BOOL := FALSE;
END_VAR
	MemFnc 													:= FNC_RUN;
	THIS^.Execute											:= Execute;
	
IF NOT __ISVALIDREF(rAxis) 
THEN
	Busy													:= NOT Error;
	ErrorId													:= E_AdsErr.DEVICE_INVALIDPARM;
	Error													:= TRUE;
	Done													:= FALSE;
	CmdAborted												:= FALSE;
	MemFnc													:= SEL(Execute , -1 ,MemFnc); 
	RETURN;
END_IF

	MC_TouchProbe(
		Execute			:= Execute,
		WindowOnly		:= WindowOnly,
		FirstPosition	:= FirstPosition,
		LastPosition	:= LastPosition,
		Axis			:= rAxis,
		TriggerInput	:= TriggerInput,
		Done			=> Done,
		Busy			=> Busy,
		CommandAborted	=> CmdAborted,
		Error			=> Error,
		ErrorID			=> ErrorID,
		RecordedPosition=> RecordedPosition,
		RecordedData 	=> RecordedData);

	IF NOT Execute AND NOT Busy
	THEN
		MemFnc												:= -1;
	END_IF
	
	run														:= busy;
END_METHOD

END_FUNCTION_BLOCK

// POUs/Motion/TF50xx-NC/03_Utilities/AX_JOB
FUNCTION_BLOCK AX_JOB (* Datatyp/Object - Ax Start data *)
VAR_INPUT
//	name						:	STRING(10);
	Fnc														:	INT := 0;
	BufferMode												:	MC_BufferMode := MC_Aborting;(* 	MC_Aborting,
																									MC_Buffered,
																									MC_BlendingLow,
																									MC_BlendingPrevious,
																									MC_BlendingNext,
																									MC_BlendingHigh *)
	Direction												:	MC_Direction := MC_POSITIVE_DIRECTION;	(*	MC_POSITIVE_DIRECTION,
																						   					MC_SHORTeSTATE.WAY,
																						   					MC_NEGATIVE_DIRECTION,
																						   					MC_CURRENT_DIRECTION *)
	Target													:	LREAL	:= 0.0; // target position
	Velo													: 	LREAL	:= 0.0; // target velocity mm/s
	Override												:	LREAL := 100.0; // override
	Acc														:	LREAL := 0.0; // acceleration
	Dec														:	LREAL := 0.0; // deceleration
	Jerk													:	LREAL := 0.0; // jerk
	InTarget												:	BOOL := FALSE;
	InPosWindow												:	BOOL := FALSE;
END_VAR
VAR_OUTPUT
END_VAR
VAR
END_VAR

;

METHOD PUBLIC reset : BOOL
VAR_INPUT
END_VAR
Fnc															:= 0;
BufferMode													:= MC_Aborting;
Direction													:= MC_CURRENT_DIRECTION;
Target														:= 0;
Velo														:= 0;
Override													:= 0;
InTarget													:= FALSE;
InPosWindow													:= FALSE;
reset														:= TRUE;
END_METHOD

END_FUNCTION_BLOCK

// POUs/Motion/TF50xx-NC/03_Utilities/AxAutoFct
{attribute 'no_check'}
FUNCTION_BLOCK AxAutoFct
VAR_INPUT
	Enable													:	BOOL := FALSE;(* Enable block *)
	AutoInit												:	BOOL := TRUE; (* TRUE=With Enable force status will be written to axis / FALSE=Force values will only be written on change *) 
	AxisId													: 	DWORD; (* ID der Achse *)
	ForceSoftLimit											:	BOOL := TRUE; (* TRUE => SoftLimitMonitoring = True *)
	ForceCalibration										:	BOOL := FALSE;(* TRUE => Calibrated = True  *)
	ForcePosLagMon											:	BOOL := TRUE; (* TRUE => Position Lag Monitoring = True  *)
	ForcePosMon												:	BOOL := TRUE; (* TRUE => In Position Monitoring = True  *)
	ForceTargetMon											:	BOOL := TRUE; (* TRUE => In Target Monitoring = True  *)
END_VAR                         							
VAR_IN_OUT                      							
END_VAR                         							
VAR_OUTPUT        
	{attribute 'displaymode':='binary'}              							
	Status													:	BYTE := 0;
	Busy													:	BOOL := FALSE;
	Error													:	BOOL := FALSE;
	ErrorID													:	UDINT := 0;
END_VAR                         	

VAR
(* Cache **********************************************************************)
	State													: 	INT;
	InitDone												:	BYTE;
	LastErrText												:	STRING(20);
	
(* Instances *******************************************************************)
	WriteAdsPara											: 	ADSWRITE := (NetID:= '' , Port:=AMSPORT_R0_NC, TmOut	:= DEFAULT_ADS_TIMEOUT);

(* Dummy  *********************************************************************)
	tmpWORD													:	UINT;

END_VAR

	(* Enable/Disable of: Soft limit monitoring, Target monitoring, Pos. Lag monitoring,  Calibration 	*)
	(*																									*)
	(****************************************************************************************************)

(* writing parameters *******************************************************************************)
IF NOT Enable 
THEN
	Status.0 												:= NOT forceSoftLimit;
	Status.1 												:= NOT forceCalibration;
	Status.2 												:= NOT forcePosLagMon;
	Status.3 												:= NOT forcePosMon;
	Status.4 												:= NOT forceTargetMon;
	            											
	InitDone 												:= SEL(AutoInit , 2#0001_1111 , 2#0000_0000);
                											
	State 													:= 0;
	Error													:= FALSE;
	ErrorID													:= 0;
	Busy 													:= FALSE;
ELSIF AxisId = 0 
THEN
	ErrorID													:= E_AdsErr.DEVICE_INVALIDPARM;
	Error													:= FALSE;
	Busy													:= FALSE;
ELSE
	CASE State OF
	0:	(* Init *)

		Busy := FALSE;

		IF NOT WriteAdsPara.BUSY
			AND NOT WriteAdsPara.WRITE
		 	AND NOT Error
		THEN
			IF (forceSoftLimit XOR status.0) OR NOT InitDone.0 THEN
				InitDone.0 									:= TRUE;
				status.0 									:= forceSoftLimit;
				tmpWord 									:= BOOL_TO_UINT(forceSoftLimit);
				State 										:= 1;
				Busy 										:= TRUE;

			ELSIF(forceCalibration XOR status.1) OR NOT InitDone.1 THEN
				InitDone.1 									:= TRUE;
				status.1 									:= forceCalibration;
				tmpWord 									:= BOOL_TO_UINT(forceCalibration);
				State 										:= 10;
				Busy 										:= TRUE;
	
			ELSIF(forcePosLagMon XOR status.2) OR NOT InitDone.2 THEN
				InitDone.2 									:= TRUE;
				status.2 									:= forcePosLagMon;
				tmpWord 									:= BOOL_TO_UINT(forcePosLagMon);
				State 										:= 20;
				Busy 										:= TRUE;
			ELSIF(forcePosMon XOR status.3) OR NOT InitDone.3 THEN
				InitDone.3 									:= TRUE;
				status.3 									:= forcePosMon;
				tmpWord 									:= BOOL_TO_UINT(forcePosMon);
				State 										:= 30;
				Busy 										:= TRUE;
			ELSIF(forceTargetMon XOR status.4) OR NOT InitDone.4 THEN
				InitDone.4 									:= TRUE;
				status.4 									:= forceTargetMon;
				tmpWord 									:= BOOL_TO_UINT(forceTargetMon);
				State 										:= 40;
				Busy 										:= TRUE;
		
			END_IF
		ELSE
			WriteAdsPara	(Write := FALSE);
		END_IF

	1: (* toggle positive limit switches ****************************************************************)
		IF NOT WriteAdsPara.Busy
			AND WriteAdsPara.Write
		THEN
			IF WriteAdsPara.Err THEN
				State 										:= 9999;  // goto Error-state 
			ELSE           									
				State 										:= State + 1;
			END_IF         	
		END_IF

		WriteAdsPara(
			IdxGrp	:=16#4000+AxisId,
			IdxOffs	:=16#1000C,
			LEN		:=SIZEOF(tmpWord),
			SrcAddr	:=ADR(tmpWord),
			Write 	:= State = 1);

	2: (* toggle negative limit switches *****************************************************************)
		IF NOT WriteAdsPara.Busy
			AND WriteAdsPara.Write
		THEN
			IF WriteAdsPara.Err THEN
				State 										:= 9999; // goto Error-state 
			ELSE
				State 										:= 99; // done 
			END_IF
		END_IF

		WriteAdsPara(
			IdxGrp	:=16#4000+AxisId,
			IdxOffs	:=16#1000B,
			LEN		:=SIZEOF(tmpWord),
			SrcAddr	:=ADR(tmpWord),
			Write 	:= State = 2);

	10: (* set referenceflag *****************************************************************)
		IF NOT WriteAdsPara.Busy
			AND WriteAdsPara.Write
		THEN
			IF WriteAdsPara.Err THEN
				State 										:= 9999;  	// goto Error-state 
			ELSE           									
				State 										:= 99; 		// done 
			END_IF
		END_IF

		WriteAdsPara(
			IdxGrp	:=16#5100+AxisId,
			IdxOffs	:=16#9,
			LEN		:=SIZEOF(tmpWord),
			SrcAddr	:=ADR(tmpWord),
			Write 	:= State = 10 );
			
	20: (* lagdistance monitoring *****************************************************************)
		IF NOT WriteAdsPara.Busy
			AND WriteAdsPara.Write
		THEN
			IF WriteAdsPara.Err THEN
				State 										:= 9999;  	// goto Error-state 
			ELSE           									
				State 										:= 99; 		// done
			END_IF
		END_IF

		WriteAdsPara(
			IdxGrp	:=16#6000+AxisId,
			IdxOffs	:=16#10,
			LEN		:=SIZEOF(tmpWord),
			SrcAddr	:=ADR(tmpWord),
			Write 	:= State = 20);
			
	30: (* Position Monitoring *****************************************************************)
		IF NOT WriteAdsPara.Busy
			AND WriteAdsPara.Write
		THEN
			IF WriteAdsPara.Err THEN
				State 										:= 9999;  	// goto Error-state 
			ELSE           									
				State 										:= 99; 		// done
			END_IF
		END_IF

		WriteAdsPara(

			IdxGrp	:=16#4000+AxisId,
			IdxOffs	:=16#F,
			LEN		:=SIZEOF(tmpWord),
			SrcAddr	:=ADR(tmpWord),
			Write 	:= State = 30 );

	40: (* Target Monitoring *****************************************************************)
		IF NOT WriteAdsPara.Busy
			AND WriteAdsPara.Write
		THEN
			IF WriteAdsPara.Err THEN
				State 										:= 9999;  	// goto Error-state 
			ELSE           									
				State 										:= 99; 		// done
			END_IF
		END_IF

		WriteAdsPara(
			IdxGrp	:=16#4000+AxisId,
			IdxOffs	:=16#15,
			LEN		:=SIZEOF(tmpWord),
			SrcAddr	:=ADR(tmpWord),
			Write 	:= State = 40 );
			
	ELSE (* case else *)
		IF WriteAdsPara.ERR THEN
			Error											:= TRUE;
			ErrorID											:= WriteAdsPara.ERRID;
			LastErrText										:= CONCAT('Err WriteAdsPara ID: ', UDINT_TO_STRING(ErrorID));
		ELSE            									
			State 											:= 0;
		END_IF
	END_CASE
END_IF

(************************************************************************************************************************)

END_FUNCTION_BLOCK

// POUs/Motion/TF50xx-NC/03_Utilities/AxAutoWriteSoftLimit
{attribute 'no_check'}
FUNCTION_BLOCK AxAutoWriteSoftLimit
VAR_INPUT
	Enable													:	BOOL := FALSE; (* Enable Block *)
	AxId													: 	DWORD; (* ID der Achse *)
	SoftLimitPos											:	LREAL;
	SoftLimitNeg											:	LREAL;
END_VAR                         							
VAR_IN_OUT                      							
END_VAR                         							
VAR_OUTPUT        
	Busy													:	BOOL := FALSE;
	Error													:	BOOL := FALSE;
	{attribute 'displaymode':='hex'}  
	ErrorID													:	UDINT := 0;
END_VAR                         	
VAR
(* Cache **********************************************************************)
	State													: 	INT;
	MemLimitPos												:	LREAL;
	MemLimitNeg												:	LREAL;
	WriteReg												:	BYTE;

(* Instances *******************************************************************)
	WriteAdsPara											: 	ADSWRITE := (NetId	:= '' , Port := 500, TmOut	:= DEFAULT_ADS_TIMEOUT);

(* Dummy  *********************************************************************)
END_VAR

	(* Easy soft limit change 																		*)
	(************************************************************************************************)

(* writing parameters *******************************************************************************)
IF NOT Enable 
THEN
	MemLimitPos												:= SoftLimitPos;
	MemLimitNeg												:= SoftLimitNeg;
	                										
	State 													:= 0;
	Error													:= FALSE;
	ErrorID													:= 0;
	Busy 													:= FALSE;
ELSIF Axid = 0 
THEN
	ErrorID													:= E_AdsErr.DEVICE_INVALIDPARM;
	Error													:= FALSE;
	Busy													:= FALSE;
ELSE
	CASE State OF
	0:	(* Init *)

		Busy 												:= FALSE;

		IF NOT WriteAdsPara.BUSY
			AND NOT WriteAdsPara.WRITE
		 	AND NOT Error
		THEN
			WriteReg.0										:= SoftLimitPos <> MemLimitPos;
			WriteReg.1										:= SoftLimitNeg <> MemLimitNeg;
			
			IF WriteReg <> 0
			THEN
				Busy 										:= TRUE;
				state										:= state + SEL(WriteReg.0, 2, 1); //Jump to 2 if only negative changed
				MemLimitPos									:= SoftLimitPos;
				MemLimitNeg									:= SoftLimitNeg;
			END_IF
		ELSE
			WriteAdsPara	(Write := FALSE);
		END_IF

	1: (* Write positive limit to NC ****************************************************************)
		WriteAdsPara( Write := WriteReg.0, IdxGrp	:=16#4000+AxID, IdxOffs	:=16#1000E, LEN	:=SIZEOF(MemLimitPos), SrcAddr	:=ADR(MemLimitPos));	
		IF NOT WriteAdsPara.Busy
		THEN
			IF WriteAdsPara.Err 
			THEN
				ErrorId										:= WriteAdsPara.ERRID;
				Error										:= TRUE;
				Busy										:= FALSE;
				state										:= 0;
			ELSE           									
				State 										:= State + 1;
			END_IF   
			WriteAdsPara(Write := FALSE);      	
		END_IF


	2: (* Write negative limit to NC ****************************************************************)
		WriteAdsPara( Write := WriteReg.1, IdxGrp	:=16#4000+AxID, IdxOffs	:=16#1000D, LEN	:=SIZEOF(MemLimitNeg), SrcAddr	:=ADR(MemLimitNeg));	
		IF NOT WriteAdsPara.Busy
		THEN
			IF WriteAdsPara.Err 
			THEN
				ErrorId										:= WriteAdsPara.ERRID;
				Error										:= TRUE;
				Busy										:= FALSE;
				state										:= 0;
			ELSE           									
				State 										:= 0;
			END_IF   
			WriteAdsPara(Write := FALSE);      	
		END_IF
	END_CASE
END_IF

(************************************************************************************************************************)

END_FUNCTION_BLOCK

// POUs/Motion/TF50xx-NC/03_Utilities/AxCalcPosBias
{attribute 'no_check'}
//Calculates (new) NC axis position bias  
FUNCTION_BLOCK AxCalcPosBias EXTENDS FbBase
VAR_OUTPUT CONSTANT
//option settings 
	{attribute 'displaymode':='binary'}
	OPTION_WRITE_TO_NC										: 	BYTE :=2#0000_0001; //New position offset (bias) will directly written into the NC
END_VAR
VAR_INPUT
	{attribute 'displaymode':='binary'}
	Options													:	BYTE := 2#0000_0000; (* option constants are predefined, so they can accordingly be passed symbolically to the block *)
	SetPos													: 	LREAL := 0.0; //New actual positon of axis 
END_VAR
VAR_IN_OUT
	Axis													:	AXIS_REF;
END_VAR
VAR_OUTPUT
	RawPos													: LREAL; // Uncorrected axis position (Offset = 0.0)	
	Offset													: LREAL; // New postition offset (Position bias) 

END_VAR
VAR
(*  Memory *****************************************************)
	LastErrorId												:	UDINT;
	LastErrorState											:	INT;

(*  Timer ******************************************************)


(*  Trigger ****************************************************)

(*  Blocks *****************************************************)
	ReadAdsPara												: ADSREAD := (NetID:= '' , Port:=AMSPORT_R0_NC,TmOut := DEFAULT_ADS_TIMEOUT );
	WriteAdsPara											: ADSWRITE := (NetID:= '' , Port:=AMSPORT_R0_NC,TmOut := DEFAULT_ADS_TIMEOUT );

(*  Error ******************************************************)
(*  Dummys *****************************************************)
	{attribute 'hide' := ''}
END_VAR

	(* Calculate new pos bias (position offset)			 	 *)
	(*********************************************************)
	
(* Sequence ********************************************************)

	rtExecute(CLK := Execute);
	CASE state OF
	0 : 
		Busy 												:= FALSE;
		IF NOT Execute THEN
			Done 											:= FALSE;
			Error 											:= FALSE;
			ErrorID 										:= 0;
		END_IF
		IF rtExecute.Q THEN
			ReadAdsPara( Read := FALSE ); 
			WriteAdsPara(Write := FALSE);
			Busy											:= TRUE;
			Offset											:= 0.0;
			RawPos											:= 0.0;
			Done 											:= FALSE;
			Error 											:= FALSE;
			ErrorID 										:= 0;
			state 											:= state + 1;
		END_IF
		
		
	(* Read current pos. bias **********************************************)
	1:
		ReadAdsPara(Read:= TRUE,	IDxGrp:=(16#5000+Axis.NcToPlc.AxisId) , IDxOffs:=16#7,LEN:=SIZEOF(Offset), DestAddr:=ADR(Offset));	
		IF NOT ReadAdsPara.BUSY
		THEN
			IF ReadAdsPara.ERR
			THEN
				Busy										:= FALSE;
				Error										:= TRUE;
				ErrorID										:= ReadAdsPara.ERRID;
				LastErrorState								:= state;
				LastErrorId									:= ErrorId;
				state										:= 0;
			ELSE //Calculate new Pos bias
				RawPos										:= Axis.NcToPlc.ActPos - Offset;	
				Offset										:= SetPos - RawPos;
				IF (OPTION_WRITE_TO_NC AND Options) > 0
				THEN
					state									:= state + 1;
				ELSE
					Busy									:= FALSE;
					Done									:= TRUE;
					state									:= 0;					
				END_IF
			END_IF
		END_IF
		
	2:
		WriteAdsPara(Write:= TRUE,	IDxGrp:=(16#5000+Axis.NcToPlc.AxisId) , IDxOffs:=16#7,LEN:=SIZEOF(Offset), SrcAddr:=ADR(Offset));	
		IF NOT WriteAdsPara.BUSY
		THEN
			IF WriteAdsPara.ERR
			THEN
				Busy										:= FALSE;
				Error										:= TRUE;
				ErrorID										:= WriteAdsPara.ERRID;
				LastErrorId									:= ErrorId;
				LastErrorState								:= state;
				state										:= 0;
			ELSE			
				Busy										:= FALSE;
				Done										:= TRUE;
				state										:= 0;					
			END_IF
		END_IF		
	END_CASE

(****************************************************************************************)

PROPERTY PUBLIC optWritePosBiasToNC : BOOL
GET
optWritePosBiasToNC := Options.0;
END_GET
SET
Options.0 := optWritePosBiasToNC;
END_SET
END_PROPERTY

END_FUNCTION_BLOCK

// POUs/Motion/TF50xx-NC/03_Utilities/AxSoftSyncDistance
//Use this FB if NC-Reference mode is set to "Software Sync" or "Hardware-Sync".
//It is mandatory that the NC encoder parameter "Encoder Sub Mask (absolute range maximum value)" is set to the correct value!
//
//This FB checks the disctance between the falling edge of an reference sensor 
//and the final reference flag of the encoder (e.g. SingleTurn overflow in mode SoftwareSync)
//In case these two signals are very close together, it might be possible that the reference position varied about one motor turn
//depending whether the falling edge of the reference sensor occured before or after the software sync impulse.
//
//The FB reports an OK if the resulting distance if greater or equel than the "MinDistanceInDeg". 
{attribute 'no_check'}
FUNCTION_BLOCK AxSoftSyncDistance EXTENDS FbBase
VAR_OUTPUT CONSTANT
//option settings 
END_VAR
VAR CONSTANT
	DEG_PER_TURN											:	LREAL := 360.0;	
END_VAR
VAR_INPUT
	MinDistanceInDeg										:	LREAL := 45.0; //Minmum required distance between falling edge of sensor and software sync reference impuls (Single turn overflow)   
END_VAR
VAR_IN_OUT
	Axis													:	AXIS_REF;
END_VAR
VAR_OUTPUT
	Distance												: LREAL; //In user units (e.g. mm)
	DistancePerTurn											: LREAL; //In user units (e.g. mm)
	DistanceInDeg											: LREAL; //Resulting distance in degrees	
	OK														: BOOL;  //Inidcates whether the distance between falling edge of sensor and software sync is greater or equal than MinDistanceInDeg  
END_VAR
VAR
(*  Memory *****************************************************)
	LastErrorState											:	INT;
	LastErrorId												:	UDINT;
	ScalingNumerator										:	LREAL;
	ScalingDenumerator										:	LREAL;
	Scaling													:	LREAL;
	RefSystem												:	UDINT;
	RefMode													:	UDINT;
	{attribute 'displaymode':='hex'}
	EncSubMask												:	UDINT;


(*  Timer ******************************************************)

(*  Trigger ****************************************************)

(*  Blocks *****************************************************)
	ReadAdsPara												: ADSREAD := (NetID:= '' , Port:=AMSPORT_R0_NC,TmOut := DEFAULT_ADS_TIMEOUT );

(*  Error ******************************************************)
(*  Dummys *****************************************************)
	{attribute 'hide' := ''}
END_VAR

	(* Check distance between falling edge of reference sensor and deteced sync impulse		*)
	(****************************************************************************************)
	
(* Sequence ********************************************************)
	rtExecute(CLK := Execute);
	CASE state OF
	0 : 
		Busy 												:= FALSE;
		IF NOT Execute THEN
			OK												:= FALSE;
			Done 											:= FALSE;
			Error 											:= FALSE;
			ErrorID 										:= 0;
		END_IF
		IF rtExecute.Q THEN
			ReadAdsPara( Read := FALSE); 
			Busy											:= TRUE;
			Distance										:= 0.0;
			ScalingNumerator								:= 0.0;
			ScalingDenumerator								:= 0.0;
			Scaling											:= 0.0;
			RefSystem										:= 0;
			EncSubMask										:= 0;
			OK												:= FALSE;
			Done 											:= FALSE;
			Error 											:= FALSE;
			ErrorID 										:= 0;
			state 											:= state + 1;
		END_IF
		
		
	(* Read scaling numerator **********************************************)
	1:
		ReadAdsPara(Read:= TRUE,	IDxGrp:=(16#5000+Axis.NcToPlc.AxisId) , IDxOffs:=16#23,LEN:=SIZEOF(ScalingNumerator), DestAddr:=ADR(ScalingNumerator));	
		IF NOT ReadAdsPara.BUSY
		THEN
			IF ReadAdsPara.ERR
			THEN
				Busy										:= FALSE;
				Error										:= TRUE;
				ErrorID										:= ReadAdsPara.ERRID;
				LastErrorState								:= state;
				LastErrorId									:= ErrorId;
				state										:= 0;
			ELSE 
				state										:= state + 1;						
			END_IF
			ReadAdsPara( Read := FALSE);
		END_IF
		
	(* Read scaling denumerator **********************************************)
	2:
		ReadAdsPara(Read:= TRUE,	IDxGrp:=(16#5000+Axis.NcToPlc.AxisId) , IDxOffs:=16#24,LEN:=SIZEOF(ScalingDenumerator), DestAddr:=ADR(ScalingDenumerator));	
		IF NOT ReadAdsPara.BUSY
		THEN
			IF ReadAdsPara.ERR
			THEN
				Busy										:= FALSE;
				Error										:= TRUE;
				ErrorID										:= ReadAdsPara.ERRID;
				LastErrorState									:= state;
				LastErrorId									:= ErrorId;
				state										:= 0;
			ELSE
				Scaling										:= ScalingNumerator / SEL(ScalingDenumerator = 0.0, ScalingDenumerator , 1.0);	
				IF Scaling = 0.0
				THEN
					Busy									:= FALSE;
					Error									:= TRUE;
					ErrorID									:= MC_ERROR_PARAMETER_NOT_CORRECT;
					LastErrorState								:= state;
					LastErrorId									:= ErrorId;
					state									:= 0;	
				ELSE
					state									:= state + 1;
				END_IF					
			END_IF
			ReadAdsPara( Read := FALSE);
		END_IF

	(* Read distance in user units **********************************************)
	3:
		ReadAdsPara(Read:= TRUE,	IDxGrp:=(16#5100+Axis.NcToPlc.AxisId) , IDxOffs:=16#101,LEN:=SIZEOF(Distance), DestAddr:=ADR(Distance));	
		IF NOT ReadAdsPara.BUSY
		THEN
			IF ReadAdsPara.ERR
			THEN
				Busy										:= FALSE;
				Error										:= TRUE;
				ErrorID										:= ReadAdsPara.ERRID;
				LastErrorState									:= state;
				LastErrorId									:= ErrorId;
				state										:= 0;
			ELSE 
				state										:= state + 1;			
			END_IF
			ReadAdsPara( Read := FALSE);
		END_IF
		
	(* Read selected reference system **********************************************)
	4:
		ReadAdsPara(Read:= TRUE,	IDxGrp:=(16#5000+Axis.NcToPlc.AxisId) , IDxOffs:=16#19,LEN:=SIZEOF(RefSystem), DestAddr:=ADR(RefSystem));	
		IF NOT ReadAdsPara.BUSY
		THEN
			IF ReadAdsPara.ERR
			THEN
				Busy										:= FALSE;
				Error										:= TRUE;
				ErrorID										:= ReadAdsPara.ERRID;
				LastErrorState									:= state;
				LastErrorId									:= ErrorId;
				state										:= 0;
			ELSE 
				state										:= state + 1;					
			END_IF
			ReadAdsPara( Read := FALSE);
		END_IF
	
	(* Read selected reference mode **********************************************)
	5:
		ReadAdsPara(Read:= TRUE,	IDxGrp:=(16#5000+Axis.NcToPlc.AxisId) , IDxOffs:=16#107,LEN:=SIZEOF(RefMode), DestAddr:=ADR(RefMode));	
		IF NOT ReadAdsPara.BUSY
		THEN
			IF ReadAdsPara.ERR
			THEN
				Busy										:= FALSE;
				Error										:= TRUE;
				ErrorID										:= ReadAdsPara.ERRID;
				LastErrorState									:= state;
				LastErrorId									:= ErrorId;
				state										:= 0;
			ELSE 
				state										:= state + 1;					
			END_IF
			ReadAdsPara( Read := FALSE);
		END_IF
	
	(* Read EncSubMask (Inc per turn) **********************************************)
	6:
		ReadAdsPara(Read:= TRUE,	IDxGrp:=(16#5000+Axis.NcToPlc.AxisId) , IDxOffs:=16#108,LEN:=SIZEOF(EncSubMask), DestAddr:=ADR(EncSubMask));	
		IF NOT ReadAdsPara.BUSY
		THEN
			IF ReadAdsPara.ERR
			THEN
				Busy										:= FALSE;
				Error										:= TRUE;
				ErrorID										:= ReadAdsPara.ERRID;
				LastErrorState									:= state;
				LastErrorId									:= ErrorId;
				state										:= 0;
			ELSIF EncSubMask = 0
			THEN
				Busy										:= FALSE;
				Error										:= TRUE;
				ErrorID										:= MC_ERROR_PARAMETER_NOT_CORRECT;
				LastErrorState									:= state;
				LastErrorId									:= ErrorId;
				state										:= 0;			
			ELSE
				state										:= state + 1;					
			END_IF
			ReadAdsPara( Read := FALSE);
		END_IF
		
	(* Check reference value ************************************)
	7:
		DistancePerTurn										:= EncSubMask * Scaling;
		DistanceInDeg										:= (DEG_PER_TURN / DistancePerTurn) * Distance;	
																		
		OK													:= ABS(DistanceInDeg) <= DEG_PER_TURN - ABS(MinDistanceInDeg)  
																AND ABS(DistanceInDeg) >= ABS(MinDistanceInDeg) ;							
	
		Busy												:= FALSE;
		Done												:= TRUE;
		state												:= 0;	
	END_CASE

(****************************************************************************************)

END_FUNCTION_BLOCK

// POUs/Motion/TF50xx-NC/03_Utilities/AxStatemodel
{attribute 'no_check'}
//based on Statemodel instance
//IMPORTANT call this functionblock after AxAdmin !!!!
FUNCTION_BLOCK AxStatemodel EXTENDS Statemodel_Unit
VAR_INPUT 
	SafetyOK												:	BOOL := TRUE; //Drive safety card OK
	ENDisableInAborting										:	BOOL := FALSE; //Disable the axis directly in aborting instead of executing MC_Stop with given emergency dynamics  
	ENSoEReset												:	BOOL := TRUE; 
	ErrorActive												:	BOOL := FALSE; //Axis in error	
	EmergencyDec											:	LREAL := 0.0; //Emergency dec used in Aborting 
	EmergencyJerk											:	LREAL := 0.0; //Emergency jekr used in Aborting 
	rAxis													:	REFERENCE TO AXIS_REF := 0;
END_VAR
VAR_OUTPUT
END_VAR
VAR
	MC_Stop													: 	MC_Stop;
	MC_Reset												:	MC_Reset;
	SOE_Reset												:	FB_SoEReset;
	Mainstate												:	INT := 0;
	Ton_Seq													:	TON;
{attribute 'displaymode':='binary'}
	MemAbortingStep											:	BYTE; //Show online reasons for the aporting steps
END_VAR

	(* Axis UnitStateCtrl				 		V1.3		*)
	(*														*)
	(********************************************************)

(* check rAxis ************************************************)
IF NOT __ISVALIDREF(rAxis) 
THEN 
(*	ErrorText			:= 'Pointer pAxis invalid (0)'; *)
	RETURN;
END_IF

(* work local sub ****************************************)
	unit.name			:= CONCAT('Unit Axis ID: ', UDINT_TO_STRING(rAxis.NcToPlc.AxisId));

(* Call super ***************************************)
	SUPER^(); //Execute generic unit
		
(*********************************************************)

METHOD PROTECTED aborted : BOOL //Return value = TRUE if execution finsihed
VAR_INPUT
END_VAR
rAxis.PlcToNc.ControlDWord.0 						:= FALSE; (* Enable *)
rAxis.PlcToNc.ControlDWord.1 						:= FALSE; (* Enable_Positive *)
rAxis.PlcToNc.ControlDWord.2 						:= FALSE; (* Enable_Negative *)

MC_Stop(
	Axis			:= rAxis,
	Execute			:= 	MC_Stop.Execute 
						AND F_AxisControlLoopClosed(stateDWord := rAxis.NcToPlc.stateDWord) 
						AND rAxis.Status.PTPmode ,  (* Block new motion cmd *)
	Deceleration	:= ,
	Jerk			:= ,
	Options			:= ,
	Done			=> ,
	Busy			=> ,
	Active			=> ,
	CommandAborted	=> ,
	Error			=> ,
	ErrorID			=> );
	
Aborted												:= MC_Stop.Done OR MC_Stop.Error OR NOT F_AxisControlLoopClosed(stateDWord := rAxis.NcToPlc.stateDWord);
END_METHOD

METHOD PROTECTED aborting : BOOL //Return value = TRUE if execution finsihed
VAR_INPUT
END_VAR
CASE Mainstate OF
		0: (* Step 1 -> start stopping *)
			MemAbortingStep									:= 0;
			IF NOT rAxis.Status.PTPmode
				OR rAxis.Status.ProtectedMode
				OR rAxis.Status.MotionCommandsLocked
				OR NOT rAxis.Status.Operational
			THEN (* axis is slave-axis *)
				Mainstate									:= 99;
				MemAbortingStep.7							:= TRUE; 
			ELSIF ENDisableInAborting
			THEN
				rAxis.PlcToNc.ControlDWord.0 				:= FALSE; (* Enable *)
				rAxis.PlcToNc.ControlDWord.1 				:= FALSE; (* Enable_Positive *)
				rAxis.PlcToNc.ControlDWord.2 				:= FALSE; (* Enable_Negative *)
				MemAbortingStep.2							:= TRUE;
				Mainstate									:= 99;	
			ELSE
				IF NOT MC_Stop.busy      					
				THEN                        					
					MemAbortingStep.1						:= TRUE;
					Mainstate								:= 99;
				END_IF

				MC_Stop(
					Axis			:= rAxis,
					Execute			:= Mainstate = 99 ,
					Deceleration	:= EmergencyDec,(* NOT-HALT Parameter uebergeben *)
					Jerk			:= EmergencyJerk, (* NOT-HALT Parameter uebergeben *)
					Options			:= ,
					Done			=> ,
					Busy			=> ,
					Active			=> ,
					CommandAborted	=> ,
					Error			=> ,
					ErrorID			=> );
			END_IF

		99: (* Step 2 -> if stopped or safety signal = FALSE *) 
			MC_Stop(
				Axis			:= rAxis,
				Execute			:= ,
				Deceleration	:= ,
				Jerk			:= ,
				Options			:= ,
				Done			=> ,
				Busy			=> ,
				Active			=> ,
				CommandAborted	=> ,
				Error			=> ,
				ErrorID			=> );

			IF NOT F_AxisControlLoopClosed(stateDWord := rAxis.NcToPlc.stateDWord)
			THEN
				MemAbortingStep.4							:= TRUE;
				Unit.StateComplete();
				Aborting									:= TRUE;			
			ELSIF MC_Stop.Execute AND rAxis.Status.NotMoving AND (MC_Stop.Done OR MC_Stop.Error)	
			THEN                        					
				MemAbortingStep.3							:= TRUE;
				Unit.StateComplete();
				Aborting									:= TRUE;
			END_IF
		END_CASE
END_METHOD

METHOD PROTECTED clearing : BOOL //Return value = TRUE if execution finsihed
VAR_INPUT
END_VAR
CASE Mainstate OF
0:
	MC_Stop(
		Axis			:= rAxis,
		Execute			:= FALSE,
		Deceleration	:= , 
		Jerk			:= , 
		Options			:= , 
		Done			=> , 
		Busy			=> , 
		Active			=> , 
		CommandAborted	=> , 
		Error			=> , 
		ErrorID			=> );
		
	IF NOT MC_Stop.Busy
	THEN
		Mainstate									:= 99;
	END_IF
				
99:
	IF NOT rAxis.PlcToNc.ControlDWord.0 (* Enable is already active *)
		OR F_AxisControlLoopClosed(stateDWord := rAxis.NcToPlc.stateDWord)
		OR ErrorActive
	THEN
		Clearing									:= TRUE;
		Unit.StateComplete();
	END_IF
			
END_CASE
END_METHOD

METHOD PROTECTED completing : Bool //Return value = TRUE if execution finsihed
VAR_INPUT
END_VAR
(* Fehler ausloesen *)
IF UNit.InCompleting
	AND NOT F_AxisHasJob(stateDWord := rAxis.NcToPlc.stateDWord)
THEN
	Unit.StateComplete();
	Completing											:= TRUE;
ELSE
	Completing 											:= Executing();
END_IF
END_METHOD

METHOD PROTECTED executing : booL
VAR_INPUT
END_VAR
(* Set statemodel to error if axis is in error *********)
IF rAxis.NcToPlc.ErrorCode <> 0 OR ErrorActive 
THEN
	IF unit.optEnableFwdMachineErrorToMaster
	THEN
		Unit.SetMachineError();
	ELSE
		Unit.SetLocalError();
	END_IF
END_IF
	
Executing 												:= Unit.isStateActive(Unit.State);
END_METHOD

METHOD PROTECTED resetting : Bool //Return value = TRUE if execution finsihed
VAR_INPUT
END_VAR
		CASE Mainstate OF
		0:
			Ton_Seq(IN := FALSE);
			
			MC_Reset(
				Axis		:= rAxis,
				Execute		:= FALSE);
				
			SOE_Reset(
				Axis		:= rAxis,
				Execute		:= FALSE);

			IF SOE_Reset.Busy
				OR MC_Reset.Busy
			THEN
				;
			ELSIF SafetyOK
			THEN
				Mainstate									:= 10;
			ELSE            								
				Mainstate									:= 1;
			END_IF          	

		1: (* Wartezeit bis Safety OK *)
			Ton_Seq(IN := TRUE, PT := T#3S);
			IF SafetyOK	
			THEN
				Mainstate									:= 2;
			ELSIF Ton_Seq.Q 
			THEN (* Karten nicht resetbar .... *)
				Ton_Seq(IN := FALSE);
				Mainstate									:= 10;
			END_IF
			

		2: (* Wartezeit nach Safety Reset *)
			Ton_Seq(IN :=TRUE, PT := T#100MS);
			IF Ton_Seq.Q
			THEN
				Ton_Seq(IN := FALSE);
				Mainstate									:= 10;
			END_IF

		10: 
			SOE_Reset(
				Axis	:= rAxis,
				Execute	:= ENSoEReset AND(rAxis.Status.Error OR rAxis.Status.DriveDeviceError));

			Mainstate										:= 11;

		11:
			SOE_Reset(Axis	:= rAxis);
			IF NOT SOE_Reset.Busy THEN
				Mainstate			:= 20;
			END_IF

		20:
			MC_Reset(
				Axis	:= rAxis,
				Execute	:= NOT rAxis.Status.ProtectedMode OR rAxis.Status.Error);

			Mainstate										:= 21;

		21:
			MC_Reset( Axis	:= rAxis);
			IF NOT MC_Reset.Busy 
			THEN
				Mainstate									:= 99;
				Ton_Seq(IN := FALSE);
			END_IF

		99:
			Ton_Seq(IN := TRUE, PT := T#3S);
			MC_Reset(
				Axis	:= rAxis,
				Execute	:= FALSE);
				
			SOE_Reset(
				Axis	:= rAxis,
				Execute	:= FALSE);

			IF NOT MC_Reset.Busy
				AND NOT SOE_Reset.Busy
				AND(Ton_Seq.Q OR NOT ErrorActive AND NOT rAxis.Status.Error) 
			THEN
				Unit.StateComplete();
				Resetting									:= TRUE;
			END_IF
		END_CASE
END_METHOD

METHOD PROTECTED starting : Bool
VAR_INPUT
END_VAR
Unit.StateComplete();
Starting													:= Executing();
END_METHOD

METHOD PROTECTED stateChanged : BOOL 
VAR_INPUT
	mode											:	eMODE;
	state											:	eSTATE;
END_VAR
	MainState 										:= 0;
END_METHOD

METHOD PROTECTED stopped : Bool //Return value = TRUE if execution finsihed
VAR_INPUT
END_VAR
		MC_Stop(
			Axis			:= rAxis,
			Execute			:= FALSE,
			Deceleration	:= ,
			Jerk			:= ,
			Options			:= ,
			Done			=> ,
			Busy			=> ,
			Active			=> ,
			CommandAborted	=> ,
			Error			=> ,
			ErrorID			=> );
			
		Stopped													:= MC_Stop.Done OR MC_Stop.Error;
END_METHOD

METHOD PROTECTED stopping : BOOL //Return value = TRUE if execution finsihed
VAR_INPUT
END_VAR
		CASE Mainstate OF
		0:
			IF NOT MC_Stop.busy
			THEN
				Mainstate									:= 1;
			END_IF		

			MC_Stop(
				Axis			:= rAxis,
				Execute			:= 	Mainstate <> 0 
									AND NOT rAxis.Status.ProtectedMode 
									AND rAxis.Status.PTPmode,
				Deceleration	:= ,
				Jerk			:= ,
				Options			:= ,
				Done			=> ,
				Busy			=> ,
				Active			=> ,
				CommandAborted	=> ,
				Error			=> ,
				ErrorID		=> );

		1:
			MC_Stop(
				Axis			:= rAxis,
				Execute			:= 	MC_Stop.Execute 
									AND NOT rAxis.Status.NotMoving 
									AND rAxis.Status.ControlLoopClosed, (* Not Moving or not Operational *)
				Deceleration	:= ,
				Jerk			:= ,
				Options			:= ,
				Done			=> ,
				Busy			=> ,
				Active			=> ,
				CommandAborted	=> ,
				Error			=> ,
				ErrorID			=> );

			IF NOT MC_Stop.Execute AND NOT MC_Stop.Busy
			THEN
				Mainstate									:= 99;				
			END_IF
			
		99:
			Unit.StateComplete();
			Stopping										:= TRUE;
		END_CASE
END_METHOD

END_FUNCTION_BLOCK

// POUs/Statemodel/control/Statemodel
{attribute 'no_check'}
//Mode-Statemodel controller - inspired by OMAC statemodel
//FB is able to synchronize subordinate statemodel instances as well to be a subordinate instance at the same time 
//
//				(Line control SM)
//				I				I
//			(Feeder)			(Stacker)
//			I	 	I			I		I					
//		(XYAxis) (Belts)	(XYAxis) (Belts)		
//
{attribute 'reflection'} 
FUNCTION_BLOCK Statemodel IMPLEMENTS I_Statemodel
VAR_OUTPUT CONSTANT         								
	VERSION													:	STRING(5) := 'V7';
	MIN_SLAVE												:	INT := 1;	 
	MAX_SLAVE												:	INT := PARAM.STATEMODEL_CTRL_MAX_SLAVE; //see library parameter to customize parameter	
                     
//Statemodel error codes       								
	ERROR_MACHINE											:	INT := 1;	(* Error requested in reason of fatal machine error, all subs in then same unit change their state to Stopping with error *)
	ERROR_LOCAL												:	INT := 2; 	(* Error requested from this sub *)
	ERROR_EXTERNAL											:	INT := 3; 	(* Error requested by Unit in reason of fatal machine error in other Sub *)
{attribute 'displaymode':='binary'}
	OPTION_ENABLE_MODE_SWITCH_TO_IDLE						:	BYTE := 2#0000_0001; //Mode switched to Idle automatically if state Aborted/Stopped reached - as default the mode will not change
{attribute 'displaymode':='binary'}
	OPTION_ENABLE_MODE_CHANGE_IN_EXECUTE					:	BYTE := 2#0000_0010; //Mode change in state Execute, FALSE = mode change over state stopping
{attribute 'displaymode':='binary'}
	OPTION_ENABLE_EXTERNAL_STATE_COMPLETE					:	BYTE := 2#0000_0100; //Default:Enable external use of method "StateComplete"! even if instance is controlling subs as well
{attribute 'displaymode':='binary'}	
	OPTION_DISABLE_LOCAL_ESTOP								:	BYTE := 2#0000_1000; //Disable local EStop signals, if sub ist remote controlled 
{attribute 'displaymode':='binary'}
	OPTION_ENABLE_MASCHINE_ERROR_TO_MASTER					:	BYTE := 2#0001_0000; //Default:Machine error to remote master - With FALSE, a machine error  will not further up reported to the master
{attribute 'displaymode':='binary'}
	OPTION_ENABLE_MODE_CHANGE_VIA_STATE_COMPL				:	BYTE := 2#0010_0000; //Default:Mode change over state Completing - The statemodel switches to state "Completing" as an reaction of a new SetMode
{attribute 'displaymode':='binary'}
	OPTION_ENABLE_EXPLICIT_ERROR_RESET						:	BYTE := 2#0100_0000; //Default:Hold state Stopped until error is eplicit reseted with reset - instance stays at Stopped until error will be reset, even if the remote master change into reset 
{attribute 'displaymode':='binary'}	
	OPTION_ENABLE_SET_ACT_STATE								:	BYTE := 2#1000_0000; //Enables to set actual state by property. Use with care and do not write state cyclic
END_VAR
VAR_INPUT                   							
    {attribute 'instance-path'} 
    {attribute 'noinit'} 	
	Name													:	STRING;
{attribute 'displaymode':='binary'}
	Options													:	BYTE := 	2#0000_0000
																		//	OR OPTION_ENABLE_MODE_SWITCH_TO_IDLE		//Mode switched to Idle automatically if state Aborted/Stopped reached - as default the mode will not change
																		//	OR OPTION_ENABLE_MODE_CHANGE_IN_EXECUTE		//Mode change in state Execute, FALSE = mode change over state stopping
																			OR OPTION_ENABLE_EXTERNAL_STATE_COMPLETE	//Default:Enable external use of method "StateComplete"! even if instance is controlling subs as well
																		//	OR OPTION_DISABLE_LOCAL_ESTOP				//Disable local EStop signals, if sub ist remote controlled 
																			OR OPTION_ENABLE_MASCHINE_ERROR_TO_MASTER	//Default:Machine error to remote master - With FALSE, a machine error  will not further up reported to the master
																			OR OPTION_ENABLE_MODE_CHANGE_VIA_STATE_COMPL//Default:Mode change over state Completing - The statemodel switches to state "Completing" as an reaction of a new SetMode
																			OR OPTION_ENABLE_EXPLICIT_ERROR_RESET		//Default:Hold state Stopped until error is eplicit reseted with reset - instance stays at Stopped until error will be reset, even if the remote master change into reset 
																		//	OR OPTION_ENABLE_SET_ACT_STATE				//Enables to set actual state by property. Use with care and do not write state cyclic
																			;		
(* Unit Safety Signals *)   								
	EStopDirectOK											:	BOOL := TRUE; (* -> Aborting *)
	EStopDelayOK											:	BOOL := TRUE; (* -> Aborted *)
	EStopOK													:	BOOL := TRUE; (* -> Clearing after EStop/Circuit OK *)
                            								
(* Signals *)               								
	ResetTrig												:	BOOL := FALSE; //Acknowledge/reset error - send also to subordinate instances  
	SetMode													:	eMODE := eMODE.IDLE; //Requested mode if instance is not a subordinate instance (RemotCtrlEnable = FALSE)
                            								
(* Remote UnitCtrl *)       								
	RemoteCtrlEnable										:	BOOL := TRUE;	//Statemodel follows remote master 
																						                           	
(* Sub Units - RemoteData from slave units *)
	ipSlave													:	ARRAY[MIN_SLAVE..MAX_SLAVE] OF I_Statemodel; (* RemoteData from slave units - WRITE THE ADRESS CYCLIC!! *)
END_VAR
VAR_OUTPUT
	Id														:	INT; //Unique Id for each statemodel instance
	IdRemoteMaster											:	INT; //Id of remote master 
	Info													:	STRING(30) := 'eSTATE.STARTUP'; //State name as string
	Busy													:	BOOL := TRUE; //Will be set to true as a result of a state change - set to false with method "StateComplete" to 
	SlavesInSync											:	BOOL; //local statemodel and subordinate (external) subs state are equel 
	SlavesBusy												:	BOOL; //minimum one sub is still busy - not complete
	NoOfBusySlaves											:	INT;	
	Mode													:	eMODE := eMODE.IDLE ;  //Active mode 
	State													:	eSTATE := eSTATE.STARTUP;//Active state
	EStopStartupOK											:	BOOL;	//EStop/Circuit is ok (clearing done)
	RT_StateChanged 										:	BOOL; //Rising flag to signal a state change
	(* StateBits *)         								
	InStartup												:	BOOL := TRUE; 	
	InIdle													:	BOOL ;
	InStarting												:	BOOL ;
	InStarted												:	BOOL ;
	InExecute												:	BOOL ;
	InCompleting											:	BOOL ;
	InComplete												:	BOOL ;
	InAborting												:	BOOL ;
	InAborted												:	BOOL ;
	InClearing												:	BOOL ;
	InStopping												:	BOOL ;
	InStopped												:	BOOL ;
	InResetting												:	BOOL ;
                            								   
(* optional not in use  										
	InHolding												:	BOOL := False;
	InHeld													:	BOOL := False;
	InUnholding												:	BOOL := False;
	InSuspending											:	BOOL := False;
	InSuspended												:	BOOL := False;
	InUnsuspending											:	BOOL := False;
*)       
	ErrHdl													:	ERROR_HDL;
                   								
END_VAR                     								
VAR
(* cache ********************************************)
	LastState												:	eSTATE := eSTATE.STARTUP;
	GoToAborting											:	BOOL ;
	Localreset												:	BOOL ;
	Remotereset												:	BOOL ;
	BusyIntern												:	BOOL := TRUE;
                          								
